(* CODESYS project WashingMashingProject_SimoneUtili.project

Project tree, tasks and I/O mapping:
  Device : CODESYS Control Win V3, CODESYS, version 3.5.20.0
    application Application
      libraries: Standard, 3.5.18.0 (System); VisuDialogs, * (System)
      task VISU_TASK (cyclic, interval 100 ms, priority 31) calls VisuElems.Visu_Prg
      task MainTask (cyclic, interval t#20ms, priority 1) calls ParentPolicyAutomata, Nominal_PA, WInFaulty_PA, HeatFaulty_PA, Simulation_Program, GA_Collector
      visualisation Visualization
      FUNCTIONBLOCKs/
        GAs/
          function block WaterManagement_GA [SFC]: _aSetDone_exit, _aEmptyWater_exit, _aFillWater_exit, _aInit_active, _aEmptyWater_active, _aReady_exit, _aReady_active, _aCHECKLEV_active, _aEmptyWater_entry, _aSetDone_active, _aFillWater_active, _aFillWater_entry_1
          function block TempControl_GA [SFC]: _aReady_exit, _aInit_active, _aReady_active, _aHeating_entry, _aHeating_exit, _aHeating_active
          function block DoorLocking_GA [SFC]: _aLocking_active, _aReady_active, _aInit_active, _aUnlocking_active, _aReady_exit, _aLocking_entry, _aUnlocking_entry, _aUnlocking_exit, _aLocking_exit, _aDoorCheck_active
          function block SoapEmptying_GA [SFC]: _aReady_active, _aCheckLev_active, _aReady_exit, _aInit_active, _aEmptying_active, _aEmptying_exit
          function block DrumMotor_GA [SFC]: _aBusy_active, _aReady_active, _aInit_active, _aBusy_exit
      PROGRAMs/
        program Simulation_Program [ST]
        program GA_Collector [FBD]
        Policy_Automatas/
          Child_PAs/
            program Nominal_PA [SFC]: _aCHECK_active, _aFLAGS_active, _aDoorLock_active_1, _aDoorLock_entry_1, _aDoorLock_exit_1, _aFillWater_active_1, _aFillWater_entry_1, _aFillWater_exit_1, _aTempRegON_active_1, _aStartMotor_active_1_1, _aStartMotSoap_active, _aStopMotor_active_1, _aStopMotor_exit_1, _aTempRegOFF_active_1, _aTempRegOFF_exit_1, _aEmptyWater_active_1, _aEmptyWater_exit_1, _aPhaseUpdate_active_1, _aPhaseUpdate_exit_1, _aDoorUnlock_active_1, _aDoorUnlock_exit_1, _aFinishedFlag_active_1, _aInit_active, _aDoorUnlock_entry, _aFinishedFlag_entry
            FaultManagerPAs/
              program HeatFaulty_PA [SFC]: _aDummy_exit, _aFillWater_h_active, _aMotON_h_active, _aMotON2_h_active, _aInit_exit, _aEmptyWater_h_exit, _aMotOFF_h_exit, _aPhaseUpdate_h_active, _aSoapON_h_active, _aEmptyWater_h_active, _aPhaseUpdate_h_exit, _aFillWater_h_entry, _aInit_active, _aMotOFF_h_active, _aFillWater_h_exit
              program WInFaulty_PA [SFC]: _aTempRegON_exit, _aTempOFF_w_active, _aInit_active, _aMotON_w_active, _aTempOFF_w_exit, _tLavaggio, _aStartMotor2_active, _aTempON_w_active, _aMotOFF_w_exit, _aTempON_w_entry, _aMotON2_w_entry, _tNoLavaggio, _aSoapOFF_w_exit, _aMotON2_w_active, _aSoapON_w_active, _aSoapOFF_w_active, _aMotOFF_w_active
          program ParentPolicyAutomata [SFC]: _aNominalPA_entry, _aPAController_entry, _aHLevDiagnostics_active, _aPAController_exit, _aPAUSE_Nom_active_1, _aDummy_active, _aPAUSE_Flt_active, _tMultiFaults, _tPauseRequest2, _aHeat_flt_entry, _aWaterIn_flt_entry, _aWaterIn_flt_exit, _tMultiFaults2, _aHeat_flt_exit, _tPauseRequest1, _aParentPAInit_active, _aPAController_active, _aStopHeatTest_exit, _aFillTest_active, _aPAUSE_Flt_entry, _aEmptyTest_exit, _aIDOLSTEP_entry, _aUnlockDoor_exit, _aRestore_exit, _aStartHeatTest_active, _aPAUSE_Nom_entry_1, _aFillTest_exit, _aStartHeatTest_entry, _aUnlockDoor_entry, _aIDOLSTEP_active, _aRestore_active, _aEmptyWater_exit, _aPAUSE_Nom_exit_1, _aStopHeatTest_active, _aEmptyWater_active, _aEmptyTest_active, _aFaultExpired_exit, _aPAUSE_Flt_exit, _aStartHeatTest_exit, _aUnlockDoor_active, _aNominalPA_exit, _tPauseRequest_
      FUNCTIONs/
        function SetBools [ST]
        function CheckFault [ST]
        function WMTempCheck [ST]
        function WMprogramCheck [ST]
        function FaultHMI [ST]
      Variables/
        ENUMs/
          data type WMPrograms
          data type State_FB
          data type Action_State
          data type LedStates
          data type LockerDoWhats
          data type WaterDoWhats
          data type WMTemps
          data type WInFlt_cases
          data type PolicyDegradation
          data type FaultType
          data type WashingPhase
        global variables GVL
  text list GlobalTextList
*)

// Device/Application/Variables/ENUMs/WMPrograms
//{attribute 'qualified_only'}
//{attribute 'strict'}
(*Programmi di funzionamento previsti dal comportamento nominale della lavatrice e selezionabili dall'utente*)
TYPE WMPrograms :
(
	Prelavaggio_prog := 1,
	Lavaggio_prog := 2,
	LavaggioCompleto_prog := 3
);
END_TYPE

// Device/Application/Variables/ENUMs/State_FB
//{attribute 'qualified_only'}
//{attribute 'strict'}

(*DUT enumerativo per definire lo stato presente della macchina a stati implementata nel SFC di ogni GA*)
TYPE State_FB : 
(
	S_Init := 0,
	S_Ready := 1,
	S_Busy := 2,
	S_Fault
);
END_TYPE

// Device/Application/Variables/ENUMs/Action_State
//{attribute 'qualified_only'}
//{attribute 'strict'}
(*stato della macchina a stati implementata nel SFC delle politiche durante il coordinamento di un GA*)
TYPE Action_State :
(
	Start_Action := 0,
	Wait_Compl := 1,
	SetOpOk := 2
);
END_TYPE

// Device/Application/Variables/ENUMs/LedStates
//{attribute 'qualified_only'}
//{attribute 'strict'}
(*due stati di accensione o spegnimento di un led*)
TYPE LedStates :
(
	ON := 0,
	OFF := 1
);
END_TYPE

// Device/Application/Variables/ENUMs/LockerDoWhats
//{attribute 'qualified_only'}
//{attribute 'strict'}
TYPE LockerDoWhats :
(
	Do_Locking := 0,
	Do_Unlocking :=1
);
END_TYPE

// Device/Application/Variables/ENUMs/WaterDoWhats
//{attribute 'qualified_only'}
//{attribute 'strict'}
TYPE WaterDoWhats :
(
	Do_WaterFilling := 0,
	Do_WaterEmptying := 1
);
END_TYPE

// Device/Application/Variables/ENUMs/WMTemps
//{attribute 'qualified_only'}
//{attribute 'strict'}

(*Temperature dell'acqua possibili selezionabili dall'utente*)
TYPE WMTemps :
(
	Warm30 := 30,
	Warm60 := 60,
	Warm90 := 90
);
END_TYPE

// Device/Application/Variables/ENUMs/WInFlt_cases
//{attribute 'qualified_only'}
//{attribute 'strict'}
(*variabile di uscita di interfaccia del GA di gestione dell'acqua per la fault isolation specifica dell'anomalia
WaterIn sulla base del livello di acqua presente nel cestello nel momento in cui il tubo si ottura*)
TYPE WInFlt_cases :
(
	early := 1,
	mid := 2,
	late := 3
);
END_TYPE

// Device/Application/Variables/ENUMs/PolicyDegradation
//{attribute 'qualified_only'}
//{attribute 'strict'}
(* Stato di salute della Politica in esecuzione*)
TYPE PolicyDegradation :
(
	HealthyPA := 0,
	FaultyPA := 1,
	KilledPA := 2
);
END_TYPE

// Device/Application/Variables/ENUMs/FaultType
//{attribute 'qualified_only'}
//{attribute 'strict'}
(*Tipo di fault riscontrato*)
TYPE FaultType :
(
	None := 0,
	WaterIn := 1,
	WaterOut := 2,
	Heat
);
END_TYPE

// Device/Application/Variables/ENUMs/WashingPhase
//{attribute 'qualified_only'}
//{attribute 'strict'}
(*Fasi di lavoro possibili per ogni programma di funzionamento della lavatrice*)
TYPE WashingPhase :
(
	Prelavaggio := 1,
	Lavaggio := 2,
	Risciacquo := 3,
	NOP
);
END_TYPE

// Device/Application/Variables/GVL
//{attribute 'qualified_only'}
VAR_GLOBAL
	temperature		: INT;		 	(*Sensor: current temperature of the water*)
	soaplevel		: INT; 			(*Sensor: current soap level*)
	waterlevel		: INT;			(*Sensor: current water level*)
	prog_number		: INT;			(*Input: program selected by the user*)
	temp_number		: INT; 			(*Input: temperature selected by the user*)
	run				: BOOL;			(*Input: if TRUE the washing machine works*)
	fillsoap		: BOOL; 		(*Input: if TRUE the soap tray is full*)
	bulls_eye_open	: BOOL := TRUE;	(*Input: if TRUE the door is open*)

	hot				: BOOL;			(*Actuator: if TRUE the resistor turns on*)
	motor_on		: BOOL;			(*Actuator: if TRUE the basket motor is turned on*)
	bulls_eye_lock	: BOOL;			(*Actuator: if TRUE the Door is locked*)
	emptysoap		: BOOL;			(*Actuator: if TRUE the soap tray is emptied*)
	fillwater		: BOOL;			(*Actuator: if TRUE the water is added*)
	emptywater		: BOOL;			(*Actuator: if TRUE the water is drained*)

	heat_alarm		: BOOL; 		(*Visualization: if TRUE alerts the user of the resistor fault*)
	water_in_alarm	: BOOL;			(*Visualization: if TRUE alerts the user of the water intake valve fault*)
	water_out_alarm	: BOOL; 		(*Visualization: if TRUE alerts the user of the water drain valve fault*)
	soap_alarm		: BOOL;			(*Visualization: if TRUE there is no soap*)
	prog_error		: BOOL;			(*Visualization: if TRUE the program selected is wrong*)
	temp_error		: BOOL;			(*Visualization: if TRUE the temperature selected is wrong*)
	rinse			: BOOL; 		(*Visualization: if TRUE the rinsing operation is going on*)
	prewash			: BOOL; 		(*Visualization: if TRUE the prewashing operation is going on*)
	wash			: BOOL; 		(*Visualization: if TRUE the washing operation is going on*)

	motor			: INT;			(*Only for simulation: angular position of the basket*)
	heat_fail		: BOOL;			(*Only for simulation: if TRUE the resistor cannot turn on*)
	water_in_fail	: BOOL;			(*Only for simulation: if TRUE the water intake valve is faulty*)
	water_out_fail	: BOOL;			(*Only for simulation: if TRUE the water drain valve is faulty*)
	WaterManagement_GA_0: WaterManagement_GA;
	TempControl_GA_0: TempControl_GA;
	SoapEmptying_GA_0: SoapEmptying_GA;
	DoorLocking_GA_0: DoorLocking_GA;
	DrumMotor_GA_0: DrumMotor_GA;
	SelectedProg : WMPrograms;
	SelectedTemp: WMTemps;
	Action_S: Action_State := Start_Action;
	Washing_P : WashingPhase;
	OpOk: BOOL;
	ProgDone: BOOL;
	IDOL : BOOL;
	PolicyEval: PolicyDegradation := HealthyPA; //inizializzo la policy come healthy per avere il comportamento nominale all'inizio
	WashTime: TIME;
	Do_Abort: BOOL;
END_VAR

// Device/Application/PROGRAMs/Policy_Automatas/ParentPolicyAutomata
PROGRAM ParentPolicyAutomata
VAR
	FltManag: BOOL := OpOk AND WaterManagement_GA_0.EmptyWaterOk;
	Fault: ARRAY [0..2] OF FaultType:= [None,None,None];
	RestoreTime : TIME := T#5S;
	Delay : TON;
	flashing : LedStates := ON;
	i:INT := 0;
END_VAR
(* SFC genitore per gestire l'esecuzione dei PA figli (Nominale, Faulty) e per eseguire gli step di attesa (IDOL), 
ripristino del funzionamento nominale e verifica delle riparazioni da fault*)

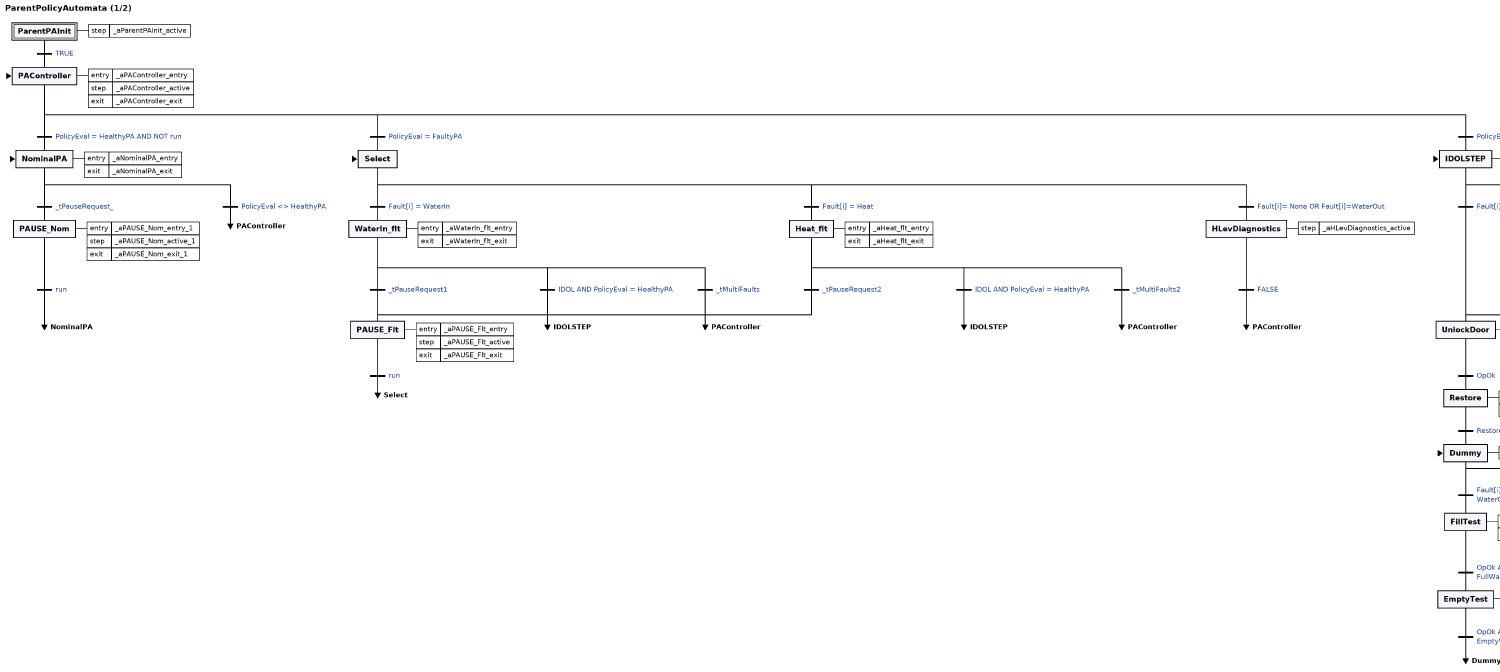
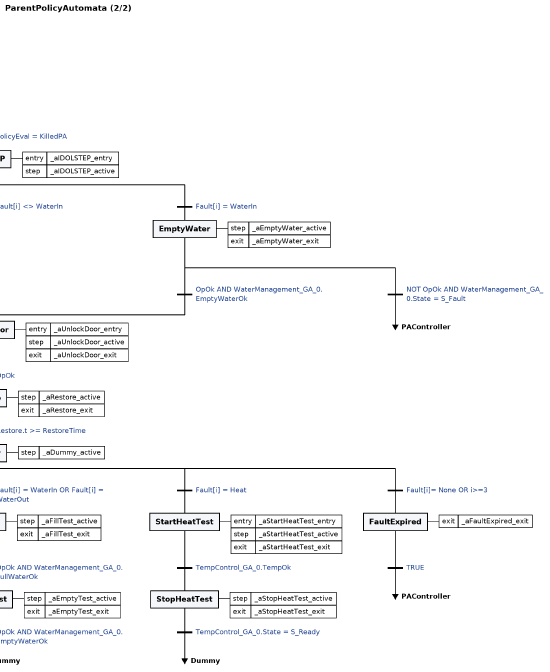
INITIAL_STEP ParentPAInit:
    _aParentPAInit_active(N);  // step action
END_STEP
TRANSITION FROM ParentPAInit TO PAController
    := TRUE;
END_TRANSITION
STEP PAController:
    _aPAController_entry(P1);  // entry action
    _aPAController_active(N);  // step action
    _aPAController_exit(P0);  // exit action
END_STEP
TRANSITION FROM PAController TO NominalPA
    := PolicyEval = HealthyPA AND NOT run;
END_TRANSITION
STEP NominalPA:
    _aNominalPA_entry(P1);  // entry action
    _aNominalPA_exit(P0);  // exit action
END_STEP
TRANSITION FROM NominalPA TO PAUSE_Nom
    := _tPauseRequest_;
END_TRANSITION
STEP PAUSE_Nom:
    _aPAUSE_Nom_entry_1(P1);  // entry action
    _aPAUSE_Nom_active_1(N);  // step action
    _aPAUSE_Nom_exit_1(P0);  // exit action
END_STEP
TRANSITION FROM PAUSE_Nom TO NominalPA
    := run;
END_TRANSITION
TRANSITION FROM NominalPA TO PAController
    := PolicyEval <> HealthyPA;
END_TRANSITION
TRANSITION FROM PAController TO Select
    := PolicyEval = FaultyPA;
END_TRANSITION
// macro FaultyPAs begins
STEP Select:
END_STEP
TRANSITION FROM Select TO WaterIn_flt
    := Fault[i] = WaterIn;
END_TRANSITION
STEP WaterIn_flt:
    _aWaterIn_flt_entry(P1);  // entry action
    _aWaterIn_flt_exit(P0);  // exit action
END_STEP
TRANSITION FROM WaterIn_flt TO PAUSE_Flt
    := _tPauseRequest1;
END_TRANSITION
TRANSITION FROM WaterIn_flt TO IDOLSTEP
    := IDOL AND PolicyEval = HealthyPA;
END_TRANSITION
TRANSITION FROM WaterIn_flt TO PAController
    := _tMultiFaults;
END_TRANSITION
TRANSITION FROM Select TO Heat_flt
    := Fault[i] = Heat;
END_TRANSITION
STEP Heat_flt:
    _aHeat_flt_entry(P1);  // entry action
    _aHeat_flt_exit(P0);  // exit action
END_STEP
TRANSITION FROM Heat_flt TO PAUSE_Flt
    := _tPauseRequest2;
END_TRANSITION
TRANSITION FROM Heat_flt TO IDOLSTEP
    := IDOL AND PolicyEval = HealthyPA;
END_TRANSITION
TRANSITION FROM Heat_flt TO PAController
    := _tMultiFaults2;
END_TRANSITION
TRANSITION FROM Select TO HLevDiagnostics
    := Fault[i]= None OR Fault[i]=WaterOut;
END_TRANSITION
STEP HLevDiagnostics:
    _aHLevDiagnostics_active(N);  // step action
END_STEP
TRANSITION FROM HLevDiagnostics TO PAController
    := FALSE;
END_TRANSITION
STEP PAUSE_Flt:
    _aPAUSE_Flt_entry(P1);  // entry action
    _aPAUSE_Flt_active(N);  // step action
    _aPAUSE_Flt_exit(P0);  // exit action
END_STEP
TRANSITION FROM PAUSE_Flt TO Select
    := run;
END_TRANSITION
TRANSITION FROM PAController TO IDOLSTEP
    := PolicyEval = KilledPA;
END_TRANSITION
// macro IdolAndTest begins
STEP IDOLSTEP:
    _aIDOLSTEP_entry(P1);  // entry action
    _aIDOLSTEP_active(N);  // step action
END_STEP
TRANSITION FROM IDOLSTEP TO UnlockDoor
    := Fault[i] <> WaterIn;
END_TRANSITION
TRANSITION FROM IDOLSTEP TO EmptyWater
    := Fault[i] = WaterIn;
END_TRANSITION
STEP EmptyWater:
    _aEmptyWater_active(N);  // step action
    _aEmptyWater_exit(P0);  // exit action
END_STEP
TRANSITION FROM EmptyWater TO UnlockDoor
    := OpOk AND WaterManagement_GA_0.EmptyWaterOk;
END_TRANSITION
TRANSITION FROM EmptyWater TO PAController
    := NOT OpOk AND WaterManagement_GA_0.State = S_Fault;
END_TRANSITION
STEP UnlockDoor:
    _aUnlockDoor_entry(P1);  // entry action
    _aUnlockDoor_active(N);  // step action
    _aUnlockDoor_exit(P0);  // exit action
END_STEP
TRANSITION FROM UnlockDoor TO Restore
    := OpOk;
END_TRANSITION
STEP Restore:
    _aRestore_active(N);  // step action
    _aRestore_exit(P0);  // exit action
END_STEP
TRANSITION FROM Restore TO Dummy
    := Restore.t >= RestoreTime;
END_TRANSITION
STEP Dummy:
    _aDummy_active(N);  // step action
END_STEP
TRANSITION FROM Dummy TO FillTest
    := Fault[i] = WaterIn OR Fault[i] = WaterOut;
END_TRANSITION
STEP FillTest:
    _aFillTest_active(N);  // step action
    _aFillTest_exit(P0);  // exit action
END_STEP
TRANSITION FROM FillTest TO EmptyTest
    := OpOk AND WaterManagement_GA_0.FullWaterOk;
END_TRANSITION
STEP EmptyTest:
    _aEmptyTest_active(N);  // step action
    _aEmptyTest_exit(P0);  // exit action
END_STEP
TRANSITION FROM EmptyTest TO Dummy
    := OpOk AND WaterManagement_GA_0.EmptyWaterOk;
END_TRANSITION
TRANSITION FROM Dummy TO StartHeatTest
    := Fault[i] = Heat;
END_TRANSITION
STEP StartHeatTest:
    _aStartHeatTest_entry(P1);  // entry action
    _aStartHeatTest_active(N);  // step action
    _aStartHeatTest_exit(P0);  // exit action
END_STEP
TRANSITION FROM StartHeatTest TO StopHeatTest
    := TempControl_GA_0.TempOk;
END_TRANSITION
STEP StopHeatTest:
    _aStopHeatTest_active(N);  // step action
    _aStopHeatTest_exit(P0);  // exit action
END_STEP
TRANSITION FROM StopHeatTest TO Dummy
    := TempControl_GA_0.State = S_Ready;
END_TRANSITION
TRANSITION FROM Dummy TO FaultExpired
    := Fault[i]= None OR i>=3;
END_TRANSITION
STEP FaultExpired:
    _aFaultExpired_exit(P0);  // exit action
END_STEP
TRANSITION FROM FaultExpired TO PAController
    := TRUE;
END_TRANSITION

ACTION _aNominalPA_entry:
WashTime := T#5S;
Nominal_PA.SFCInit := FALSE;
END_ACTION

ACTION _aPAController_entry:
IF Fault[i] <> None THEN
	i:=i+1;
END_IF
END_ACTION

ACTION _aHLevDiagnostics_active:
//Questo step rappresenta una diagnositica di alto livello di tipo A per l'interfacciamento corretto tra Politica e GA

(*Nota: questo step non dovrebbe essere mai eseguito perchè il ramo di PAFaulty viene attraversato solo nel 
caso di WaterIn o Heat fault, per nessun Fault dovrebbe essere attivo l'SFC Nominale o la fase di IdolAndStep 
nel caso di fault già gestiti*)
END_ACTION

ACTION _aPAController_exit:
FaultHMI(Fault[i], TRUE);

IF Fault[i]= None THEN
 SetBools(3,FALSE);
END_IF
END_ACTION

ACTION _aPAUSE_Nom_active_1:

END_ACTION

ACTION _aDummy_active:
//step con nessuna aziona per permettere un loop corretto dei fault nel vettore che li contiene

(*Una volta avvvenuto l'intervento di ripristino degli attuatori malfunzionanti, prima di procedere con 
un programma inserito dall'utente si fa un test delle azioni base relative all'attuatore che è stato riparato
per verificare il corretto intervento*)
END_ACTION

ACTION _aPAUSE_Flt_active:

END_ACTION

TRANSITION _tMultiFaults:
PolicyEval <> HealthyPA AND WaterManagement_GA_0.State = S_Ready
END_TRANSITION

TRANSITION _tPauseRequest2:
PolicyEval = HealthyPA AND NOT run
END_TRANSITION

ACTION _aHeat_flt_entry:
HeatFaulty_PA.SFCInit := FALSE;
TempControl_GA_0.StartTemp := FALSE;

//Le seguenti sono istruzioni per garantire un protocollo di handshake corretto tra Parent Policy e Child Policy
//Esco dallo stato di fault in modo da riconoscere un'eventuale condizione di fault aggiuntivo (fault multipli)
//durante l'esecuzione degradata del programma dovuta al primo fault
 
TempControl_GA_0.Restore := TRUE; //PER ANDARE IN READY NEL GA
WashTime := T#3S;
END_ACTION

ACTION _aWaterIn_flt_entry:
WInFaulty_PA.SFCInit := FALSE;
WaterManagement_GA_0.Restore := TRUE;
END_ACTION

ACTION _aWaterIn_flt_exit:
WInFaulty_PA.SFCPause := TRUE;

//WInFaulty_PA.SFCInit := TRUE;
WaterManagement_GA_0.Restore := FALSE;
END_ACTION

TRANSITION _tMultiFaults2:
PolicyEval <> HealthyPA AND TempControl_GA_0.State = S_Ready

//Se la politica non è più Healthy durante l'esecuzione dell'AdP HeatFaulty_PA allora
//significa che è avvenuto un altro fault
END_TRANSITION

ACTION _aHeat_flt_exit:
HeatFaulty_PA.SFCPause := TRUE;
HeatFaulty_PA.SFCInit := TRUE;
TempControl_GA_0.Restore := FALSE;
END_ACTION

TRANSITION _tPauseRequest1:
PolicyEval = HealthyPA AND NOT run
END_TRANSITION

ACTION _aParentPAInit_active:

END_ACTION

ACTION _aPAController_active:
SetBools(4,TRUE); //inizializzo le SFC Flags
IF NOT IDOL  THEN
	Fault[i] := checkFault();
END_IF
END_ACTION

ACTION _aStopHeatTest_exit:
TempControl_GA_0.StopTemp := FALSE;
i:=i+1;
END_ACTION

ACTION _aFillTest_active:
CASE Action_S OF 
Start_Action: IF WaterManagement_GA_0.State = S_Ready THEN 
				 WaterManagement_GA_0.FillTest := TRUE;
				 Action_S := Wait_Compl;
			  END_IF
			  
Wait_Compl: IF WaterManagement_GA_0.Done AND WaterManagement_GA_0.State = S_Busy THEN 
			   WaterManagement_GA_0.FillTest := FALSE;
			   Action_S := SetOpOk;
			END_IF
//protocollo di handshake di set reset del FillTest e done da parte di politica e ga per evitare attivazioni multiple
SetOpOk: IF NOT WaterManagement_GA_0.Done THEN
			OpOk := TRUE;
	     END_IF
END_CASE
END_ACTION

ACTION _aPAUSE_Flt_entry:
Do_Abort := TRUE;
SetBools(2,FALSE);
END_ACTION

ACTION _aEmptyTest_exit:
OpOk := FALSE;
Action_S := Start_Action;
i:=i+1;
END_ACTION

ACTION _aIDOLSTEP_entry:
IDOL := FALSE;
WaterManagement_GA_0.Restore := TRUE;
END_ACTION

ACTION _aUnlockDoor_exit:
OpOk := FALSE;
Action_S := Start_Action;
END_ACTION

ACTION _aRestore_exit:
SetBools(3,FALSE);
i:=0;
END_ACTION

ACTION _aStartHeatTest_active:
IF TempControl_GA_0.State = S_Ready THEN
	TempControl_GA_0.StartWhat := Warm90;
	TempControl_GA_0.HeatTest := TRUE;
END_IF
END_ACTION

ACTION _aPAUSE_Nom_entry_1:
Do_Abort := TRUE;
SetBools(2,FALSE);
END_ACTION

ACTION _aFillTest_exit:
OpOk := FALSE;
Action_S := Start_Action;
END_ACTION

ACTION _aStartHeatTest_entry:
TempControl_GA_0.StopTemp := FALSE; //protocollo di handshake per evitare attivazioni multiple
END_ACTION

ACTION _aUnlockDoor_entry:
Action_S := Start_Action;
WaterManagement_GA_0.Restore := FALSE;
END_ACTION

ACTION _aIDOLSTEP_active:
SetBools(2,FALSE); //spegnimento led fasi hmi nel caso di un fault killer
END_ACTION

ACTION _aRestore_active:
//IMPORTANTE!!
(*Questo è lo step in cui si ipotizza avvenga l'intervento da parte di un operatore esterno per eseguire la manutenzione
necessaria al ripristino del funzionamento nominale della lavatrice e delle sue funzioni, per semplicità si considera
che l'intervento avvenga senza disalimentare la lavatrice e gli attuatori stessi, nella simulazione perciò
si spengono gli switch dei fault durante questa fase caratterizzata dal lampeggiamento dei led hmi dei fault riscontrati
*)
CASE flashing OF 
ON: FaultHMI(Fault[0], FALSE);
	FaultHMI(Fault[1], FALSE);
	FaultHMI(Fault[2],FALSE);
	Delay(IN:=TRUE, PT:=T#0.3S);
	IF Delay.Q THEN
		Delay(IN:=FALSE);
		flashing := OFF;
	END_IF
OFF:FaultHMI(Fault[0], TRUE);
	FaultHMI(Fault[1], TRUE);
	FaultHMI(Fault[2],TRUE);
	Delay(IN:=TRUE, PT:=T#0.3S);
	IF Delay.Q THEN
	  Delay(IN:=FALSE); 
	  flashing := ON;
	END_IF
END_CASE
END_ACTION

ACTION _aEmptyWater_exit:
OpOk := FALSE;
Action_S := Start_Action;
END_ACTION

ACTION _aPAUSE_Nom_exit_1:
Nominal_PA.SFCPause := FALSE;
Do_Abort := FALSE;

CASE Washing_P OF 
Prelavaggio: prewash := TRUE;
Lavaggio: wash := TRUE;
Risciacquo: rinse := TRUE;
END_CASE
END_ACTION

ACTION _aStopHeatTest_active:
TempControl_GA_0.StopTemp := TRUE;
TempControl_GA_0.StartTemp := FALSE;
TempControl_GA_0.HeatTest := FALSE;
END_ACTION

ACTION _aEmptyWater_active:
(* Nel caso di fault di tipo WaterIn si è scelto di svuotare l'acqua del cestello in questo step al termine della gestione che invece risulta differenziata
a seconda del momento in cui si interrompe il riempimento*)

CASE Action_S OF 
Start_Action: IF WaterManagement_GA_0.State = S_Ready THEN 
				 WaterManagement_GA_0.Do_ := TRUE;
				 WaterManagement_GA_0.DoWhat := Do_WaterEmptying;
				 Action_S := Wait_Compl;
			  END_IF
			  
Wait_Compl: IF WaterManagement_GA_0.Done AND WaterManagement_GA_0.State = S_Busy THEN 
			   WaterManagement_GA_0.Do_ := FALSE;
			   Action_S := SetOpOk;
			ELSIF NOT WaterManagement_GA_0.Done AND WaterManagement_GA_0.State = S_Fault THEN 
				WaterManagement_GA_0.Do_ := FALSE;
				Action_S := Start_Action;
			END_IF
//protocollo di handshake di set reset del do e done da parte di politica e ga per evitare attivazioni multiple
SetOpOk: IF NOT WaterManagement_GA_0.Done THEN
			OpOk := TRUE;
	     END_IF
END_CASE
END_ACTION

ACTION _aEmptyTest_active:
CASE Action_S OF 
Start_Action: IF WaterManagement_GA_0.State = S_Ready THEN 
				 //WaterManagement_GA_0.Do_ := TRUE;
				 //WaterManagement_GA_0.DoWhat := Do_WaterEmptying;
				 WaterManagement_GA_0.EmptyTest := TRUE;
				 Action_S := Wait_Compl;
			  END_IF
			  
Wait_Compl: IF WaterManagement_GA_0.Done AND WaterManagement_GA_0.State = S_Busy THEN 
			   //WaterManagement_GA_0.Do_ := FALSE;
			   WaterManagement_GA_0.EmptyTest := FALSE;
			   Action_S := SetOpOk;
			END_IF
//protocollo di handshake di set reset del do e done da parte di politica e ga per evitare attivazioni multiple
SetOpOk: IF NOT WaterManagement_GA_0.Done THEN
			OpOk := TRUE;
	     END_IF
END_CASE
END_ACTION

ACTION _aFaultExpired_exit:
//tutti i fault sono estinti e ne è stata verificata l'assenza in seguito all'intervento dell'operatore

//inizializzo i parametri di gestione dei fault per ricominciare un altro programma di lavaggio
//della lavatrice a partire dalla Politica Nominale
i:=0;
PolicyEval := HealthyPA;
Washing_P := NOP;
Fault[0]:= None;
Fault[1]:= None;
Fault[2] := None;
END_ACTION

ACTION _aPAUSE_Flt_exit:
WInFaulty_PA.SFCPause := FALSE;
HeatFaulty_PA.SFCPause := FALSE;
Do_Abort := FALSE;

CASE Washing_P OF 
Prelavaggio: prewash := TRUE;
Lavaggio: wash := TRUE;
Risciacquo: rinse := TRUE;
END_CASE
END_ACTION

ACTION _aStartHeatTest_exit:

END_ACTION

ACTION _aUnlockDoor_active:
CASE Action_S OF 
Start_Action: IF Doorlocking_GA_0.State = S_Ready THEN 
				 Doorlocking_GA_0.Do_ := TRUE;
				 Doorlocking_GA_0.DoWhat := Do_Unlocking;
				 Action_S := Wait_Compl;
			  END_IF
			  
Wait_Compl: IF Doorlocking_GA_0.Done AND Doorlocking_GA_0.State = S_Busy THEN 
			   Doorlocking_GA_0.Do_ := FALSE;
			   Action_S := SetOpOk;
			END_IF
//protocollo di handshake di set reset del do e done da parte di politica e ga per evitare attivazioni multiple
SetOpOk: IF NOT Doorlocking_GA_0.Done THEN
			OpOk := TRUE;
	     END_IF
END_CASE
END_ACTION

ACTION _aNominalPA_exit:
Nominal_PA.SFCPause := TRUE;
END_ACTION

TRANSITION _tPauseRequest_:
PolicyEval = HealthyPA AND NOT run
END_TRANSITION

END_PROGRAM

// Device/Application/PROGRAMs/Policy_Automatas/Child_PAs/Nominal_PA
PROGRAM Nominal_PA
VAR
	TempCorrect: BOOL;
	ProgCorrect: BOOL;
	SoapCorrect: BOOL;
	LockCorrect: BOOL;
	CheckOk: BOOL;
	Delay : TON;
	flashing : LedStates := ON;
END_VAR
VAR_INPUT
	SFCInit:BOOL;
	SFCPause: BOOL;
END_VAR

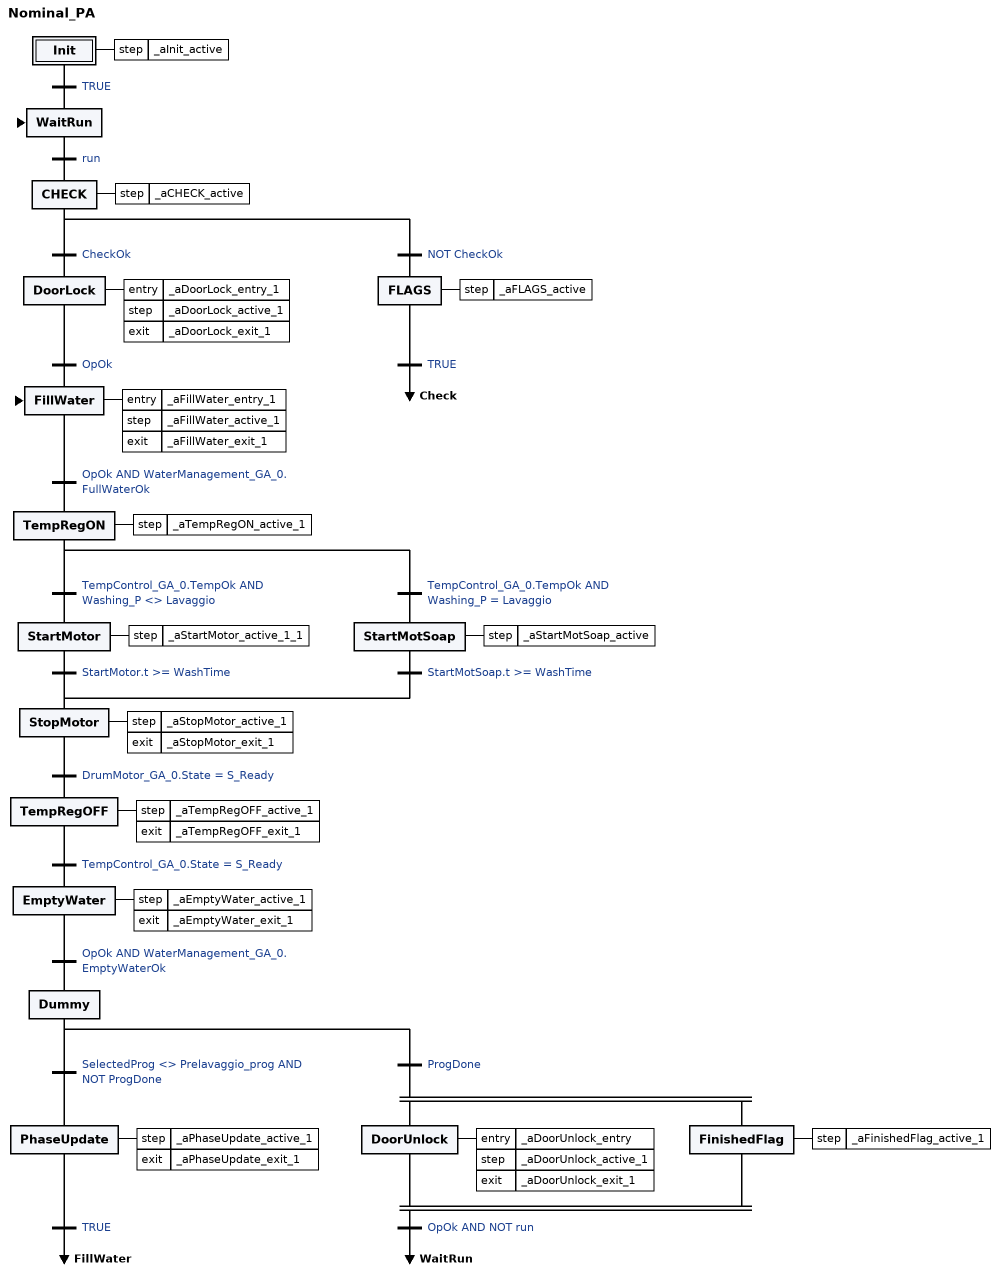
INITIAL_STEP Init:
    _aInit_active(N);  // step action
END_STEP
TRANSITION FROM Init TO WaitRun
    := TRUE;
END_TRANSITION
STEP WaitRun:
END_STEP
TRANSITION FROM WaitRun TO CHECK
    := run;
END_TRANSITION
STEP CHECK:
    _aCHECK_active(N);  // step action
END_STEP
TRANSITION FROM CHECK TO DoorLock
    := CheckOk;
END_TRANSITION
// macro WMCYCLE begins
STEP DoorLock:
    _aDoorLock_entry_1(P1);  // entry action
    _aDoorLock_active_1(N);  // step action
    _aDoorLock_exit_1(P0);  // exit action
END_STEP
TRANSITION FROM DoorLock TO FillWater
    := OpOk;
END_TRANSITION
STEP FillWater:
    _aFillWater_entry_1(P1);  // entry action
    _aFillWater_active_1(N);  // step action
    _aFillWater_exit_1(P0);  // exit action
END_STEP
TRANSITION FROM FillWater TO TempRegON
    := OpOk AND WaterManagement_GA_0.FullWaterOk;
END_TRANSITION
STEP TempRegON:
    _aTempRegON_active_1(N);  // step action
END_STEP
TRANSITION FROM TempRegON TO StartMotor
    := TempControl_GA_0.TempOk AND Washing_P <> Lavaggio;
END_TRANSITION
STEP StartMotor:
    _aStartMotor_active_1_1(N);  // step action
END_STEP
TRANSITION FROM StartMotor TO StopMotor
    := StartMotor.t >= WashTime;
END_TRANSITION
TRANSITION FROM TempRegON TO StartMotSoap
    := TempControl_GA_0.TempOk AND Washing_P = Lavaggio;
END_TRANSITION
STEP StartMotSoap:
    _aStartMotSoap_active(N);  // step action
END_STEP
TRANSITION FROM StartMotSoap TO StopMotor
    := StartMotSoap.t >= WashTime;
END_TRANSITION
STEP StopMotor:
    _aStopMotor_active_1(N);  // step action
    _aStopMotor_exit_1(P0);  // exit action
END_STEP
TRANSITION FROM StopMotor TO TempRegOFF
    := DrumMotor_GA_0.State = S_Ready;
END_TRANSITION
STEP TempRegOFF:
    _aTempRegOFF_active_1(N);  // step action
    _aTempRegOFF_exit_1(P0);  // exit action
END_STEP
TRANSITION FROM TempRegOFF TO EmptyWater
    := TempControl_GA_0.State = S_Ready;
END_TRANSITION
STEP EmptyWater:
    _aEmptyWater_active_1(N);  // step action
    _aEmptyWater_exit_1(P0);  // exit action
END_STEP
TRANSITION FROM EmptyWater TO Dummy
    := OpOk AND WaterManagement_GA_0.EmptyWaterOk;
END_TRANSITION
STEP Dummy:
END_STEP
TRANSITION FROM Dummy TO PhaseUpdate
    := SelectedProg <> Prelavaggio_prog AND NOT ProgDone;
END_TRANSITION
STEP PhaseUpdate:
    _aPhaseUpdate_active_1(N);  // step action
    _aPhaseUpdate_exit_1(P0);  // exit action
END_STEP
TRANSITION FROM PhaseUpdate TO FillWater
    := TRUE;
END_TRANSITION
TRANSITION FROM Dummy TO (DoorUnlock, FinishedFlag)
    := ProgDone;
END_TRANSITION
STEP DoorUnlock:
    _aDoorUnlock_entry(P1);  // entry action
    _aDoorUnlock_active_1(N);  // step action
    _aDoorUnlock_exit_1(P0);  // exit action
END_STEP
STEP FinishedFlag:
    _aFinishedFlag_active_1(N);  // step action
END_STEP
TRANSITION FROM (DoorUnlock, FinishedFlag) TO WaitRun
    := OpOk AND NOT run;
END_TRANSITION
TRANSITION FROM CHECK TO FLAGS
    := NOT CheckOk;
END_TRANSITION
STEP FLAGS:
    _aFLAGS_active(N);  // step action
END_STEP
TRANSITION FROM FLAGS TO Check
    := TRUE;
END_TRANSITION

ACTION _aCHECK_active:
//Per la corretta gestione dell'HMI mplementa il freeze delle variabili da hmi 
//vengono cioè salvati i primi input non più modificabili se non in un secondo ciclo di check nel programma successivo
SelectedProg := prog_number; //int to type enum
SelectedTemp := temp_number;

ProgCorrect := WMProgramCheck(SelectedProg);
TempCorrect := WMTempCheck(SelectedTemp);

IF ProgCorrect THEN
	CASE SelectedProg OF 
	Prelavaggio_prog: SoapCorrect := TRUE; //l'unico programma che non richiede il sapone è il prelavaggio perciò il check è già verificato
		Washing_P := Prelavaggio; //inilizializzazione della prima fase corrispondente al programma selezionato
		ProgDone := TRUE; //non richiede loop
		
	Lavaggio_prog: IF NOT SoapEmptying_GA_0.NoSoap THEN 
			SoapCorrect := TRUE;
		ELSE 	SoapCorrect := FALSE;
		END_IF 
	   Washing_P := Lavaggio;
	   
	LavaggioCompleto_prog: IF NOT SoapEmptying_GA_0.NoSoap THEN 
			SoapCorrect := TRUE;
		ELSE 	SoapCorrect := FALSE;
		END_IF 
	   Washing_P := Prelavaggio;
	   
	END_CASE
END_IF

IF NOT DoorLocking_GA_0.OpenDoor THEN
	LockCorrect := TRUE;
END_IF

//check delle variabili di input contemporaneamente
IF TempCorrect AND ProgCorrect AND SoapCorrect AND LockCorrect THEN 
	CheckOK := TRUE;
ELSE 
	CheckOk := FALSE;
END_IF
END_ACTION

ACTION _aFLAGS_active:
//led hmi segnalazione errore di input
soap_alarm := NOT SoapCorrect;
prog_error := NOT ProgCorrect;
temp_error := NOT TempCorrect;
END_ACTION

ACTION _aDoorLock_active_1:
CASE Action_S OF 
Start_Action: IF Doorlocking_GA_0.State = S_Ready THEN 
				 Doorlocking_GA_0.Do_ := TRUE;
				 Doorlocking_GA_0.DoWhat := Do_Locking;
				 Action_S := Wait_Compl;
			  END_IF
			  
Wait_Compl: IF Doorlocking_GA_0.Done AND Doorlocking_GA_0.State = S_Busy THEN 
			   Doorlocking_GA_0.Do_ := FALSE;
			   Action_S := SetOpOk;
			END_IF
//protocollo di handshake di set reset del do e done da parte di politica e ga per evitare attivazioni multiple
SetOpOk: IF NOT Doorlocking_GA_0.Done THEN
			OpOk := TRUE;
	     END_IF
END_CASE
END_ACTION

ACTION _aDoorLock_entry_1:
SetBools(1,FALSE); 
//spengono tutti i led di segnalazione di errori di input da hmi
//il primo parametro è il gruppo di variabili booleane da cambiare
END_ACTION

ACTION _aDoorLock_exit_1:
OpOk := FALSE;
Action_S := Start_Action;
END_ACTION

ACTION _aFillWater_active_1:
CASE Action_S OF //macchina a stati implementata con uno switch case, funziona grazie al modello di esecuzione con while intrinseco
//n.b. per fare la diagnostica di alto livello di tipo A tra politica e GA dovrei aggiungere un else nell'if per il caso il cui non si ver
//verifica mai lo stato ready(anomalia)
Start_Action: IF WaterManagement_GA_0.State = S_Ready THEN 
				 WaterManagement_GA_0.Do_ := TRUE;
				 WaterManagement_GA_0.DoWhat := Do_WaterFilling;
				 Action_S := Wait_Compl;
			  END_IF
			  
Wait_Compl: IF WaterManagement_GA_0.Done AND WaterManagement_GA_0.State = S_Busy THEN 
			   WaterManagement_GA_0.Do_ := FALSE;
			   Action_S := SetOpOk;
			   //nel caso di fault state del GA resetto il Do e inizializzo la macchina a stati
			ELSIF NOT WaterManagement_GA_0.Done AND WaterManagement_GA_0.State = S_Fault THEN 
				WaterManagement_GA_0.Do_ := FALSE;
				Action_S := Start_Action;
			END_IF
//protocollo di handshake di set reset del do e done da parte di politica e ga per evitare attivazioni multiple
SetOpOk: IF NOT WaterManagement_GA_0.Done THEN
			OpOk := TRUE;
	     END_IF
END_CASE
END_ACTION

ACTION _aFillWater_entry_1:

	CASE Washing_P OF 
	Prelavaggio: prewash := TRUE;
	Lavaggio: wash := TRUE;
	Risciacquo: rinse := TRUE;
	END_CASE
END_ACTION

ACTION _aFillWater_exit_1:
OpOk := FALSE;
Action_S := Start_Action;
END_ACTION

ACTION _aTempRegON_active_1:
IF TempControl_GA_0.State = S_Ready THEN
	TempControl_GA_0.StartWhat := SelectedTemp;
	TempControl_GA_0.StartTemp := TRUE;
END_IF
END_ACTION

ACTION _aStartMotor_active_1_1:
IF DrumMotor_GA_0.State = S_Ready THEN
	DrumMotor_GA_0.StartMotor := TRUE;
END_IF
END_ACTION

ACTION _aStartMotSoap_active:
IF DrumMotor_GA_0.State = S_Ready THEN
	DrumMotor_GA_0.StartMotor := TRUE;
END_IF

IF SoapEmptying_GA_0.State = S_Ready THEN
	SoapEmptying_GA_0.StartSoap := TRUE;
END_IF
END_ACTION

ACTION _aStopMotor_active_1:
DrumMotor_GA_0.StopMotor := TRUE;
DrumMotor_GA_0.StartMotor := FALSE;

SoapEmptying_GA_0.StopSoap := TRUE;
SoapEmptying_GA_0.StartSoap := FALSE;
END_ACTION

ACTION _aStopMotor_exit_1:
DrumMotor_GA_0.StopMotor := FALSE;
SoapEmptying_GA_0.StopSoap := FALSE;
END_ACTION

ACTION _aTempRegOFF_active_1:
TempControl_GA_0.StopTemp := TRUE;
TempControl_GA_0.StartTemp := FALSE;
END_ACTION

ACTION _aTempRegOFF_exit_1:
TempControl_GA_0.StopTemp := FALSE;
END_ACTION

ACTION _aEmptyWater_active_1:
CASE Action_S OF //macchina a stati implementata con uno switch case, funziona grazie al modello di esecuzione con while intrinseco
//n.b. per fare la diagnostica di alto livello di tipo A tra politica e GA dovrei aggiungere un else nell'if per il caso il cui non si ver
//verifica mai lo stato ready(anomalia)
Start_Action: IF WaterManagement_GA_0.State = S_Ready THEN 
				 WaterManagement_GA_0.Do_ := TRUE;
				 WaterManagement_GA_0.DoWhat := Do_WaterEmptying;
				 Action_S := Wait_Compl;
			  END_IF
			  
Wait_Compl: IF WaterManagement_GA_0.Done AND WaterManagement_GA_0.State = S_Busy THEN 
			   WaterManagement_GA_0.Do_ := FALSE;
			   Action_S := SetOpOk;
			 ELSIF NOT WaterManagement_GA_0.Done AND WaterManagement_GA_0.State = S_Fault THEN 
			   WaterManagement_GA_0.Do_ := FALSE;
			   Action_S := Start_Action;
			END_IF
//protocollo di handshake di set reset del do e done da parte di politica e ga per evitare attivazioni multiple
SetOpOk: IF NOT WaterManagement_GA_0.Done THEN
			OpOk := TRUE;
	     END_IF
END_CASE
END_ACTION

ACTION _aEmptyWater_exit_1:
OpOk := FALSE;
Action_S := Start_Action;
END_ACTION

ACTION _aPhaseUpdate_active_1:
IF SelectedProg = LavaggioCompleto_prog THEN
	CASE Washing_P OF 
	Prelavaggio: Washing_P := Lavaggio;
	
	Lavaggio : Washing_P := Risciacquo;
			   ProgDone := TRUE;
	END_CASE
END_IF

IF SelectedProg = Lavaggio_prog AND Washing_P = Lavaggio THEN
	Washing_P := Risciacquo;
	ProgDone := TRUE;
END_IF
END_ACTION

ACTION _aPhaseUpdate_exit_1:
prewash := FALSE;
wash := FALSE;
rinse := FALSE;
END_ACTION

ACTION _aDoorUnlock_active_1:

CASE Action_S OF 
Start_Action: IF Doorlocking_GA_0.State = S_Ready THEN 
				 Doorlocking_GA_0.Do_ := TRUE;
				 Doorlocking_GA_0.DoWhat := Do_Unlocking;
				 Action_S := Wait_Compl;
			  END_IF
			  
Wait_Compl: IF Doorlocking_GA_0.Done AND Doorlocking_GA_0.State = S_Busy THEN 
			   Doorlocking_GA_0.Do_ := FALSE;
			   Action_S := SetOpOk;
			END_IF
//protocollo di handshake di set reset del do e done da parte di politica e ga per evitare attivazioni multiple
SetOpOk: IF NOT Doorlocking_GA_0.Done THEN
			OpOk := TRUE;
	     END_IF
END_CASE
END_ACTION

ACTION _aDoorUnlock_exit_1:
OpOk := FALSE;
ProgDone := FALSE;
Action_S := Start_Action;
END_ACTION

ACTION _aFinishedFlag_active_1:
CASE flashing OF 
ON: SetBools(2,TRUE);
	Delay(IN:=TRUE, PT:=T#1S);
	IF Delay.Q THEN
		Delay(IN:=FALSE);
		flashing := OFF;
	END_IF
OFF: SetBools(2,FALSE);
	Delay(IN:=TRUE, PT:=T#1S);
	IF Delay.Q THEN
	  Delay(IN:=FALSE); 
	  flashing := ON;
	END_IF
END_CASE
END_ACTION

ACTION _aInit_active:
Washing_P := NOP;
END_ACTION

ACTION _aDoorUnlock_entry:
Washing_P := NOP;
END_ACTION

ACTION _aFinishedFlag_entry:

END_ACTION

END_PROGRAM

// Device/Application/FUNCTIONs/WMprogramCheck
FUNCTION WMprogramCheck : BOOL
VAR_INPUT
	InputProg : WMPrograms;
END_VAR
VAR
END_VAR

WMprogramCheck := InputProg = Prelavaggio_prog OR InputProg = Lavaggio_prog OR InputProg = LavaggioCompleto_prog;

END_FUNCTION

// Device/Application/FUNCTIONs/WMTempCheck
FUNCTION WMTempCheck : BOOL
VAR_INPUT
	InputTemp: WMTemps;
END_VAR
VAR
END_VAR

WMTempCheck := InputTemp = Warm30 OR InputTemp = Warm60 OR InputTemp = Warm90;

END_FUNCTION

// Device/Application/FUNCTIONs/SetBools
FUNCTION SetBools : BOOL
VAR_INPUT
	which: INT;
	value: BOOL;
END_VAR
VAR
END_VAR

CASE which OF 
	1:  prog_error := value;
		temp_error := value;
		soap_alarm := value;
		
	2:  prewash := value;
		wash := value;
		rinse := value;
		
	3:  water_in_alarm := value;
		water_out_alarm := value;
		heat_alarm := value;
		
	4:	Nominal_PA.SFCInit := value;
		WInFaulty_PA.SFCInit := value;
		HeatFaulty_PA.SFCInit := value;
		Nominal_PA.SFCPause := NOT value;
		WINFaulty_PA.SFCPause := NOT value;
		HeatFaulty_PA.SFCPause := NOT value;
	
END_CASE

END_FUNCTION

// Device/Application/PROGRAMs/Policy_Automatas/Child_PAs/FaultManagerPAs/WInFaulty_PA
PROGRAM WInFaulty_PA
VAR
END_VAR
VAR_INPUT
	SFCInit:BOOL;
	SFCPause: BOOL;
END_VAR

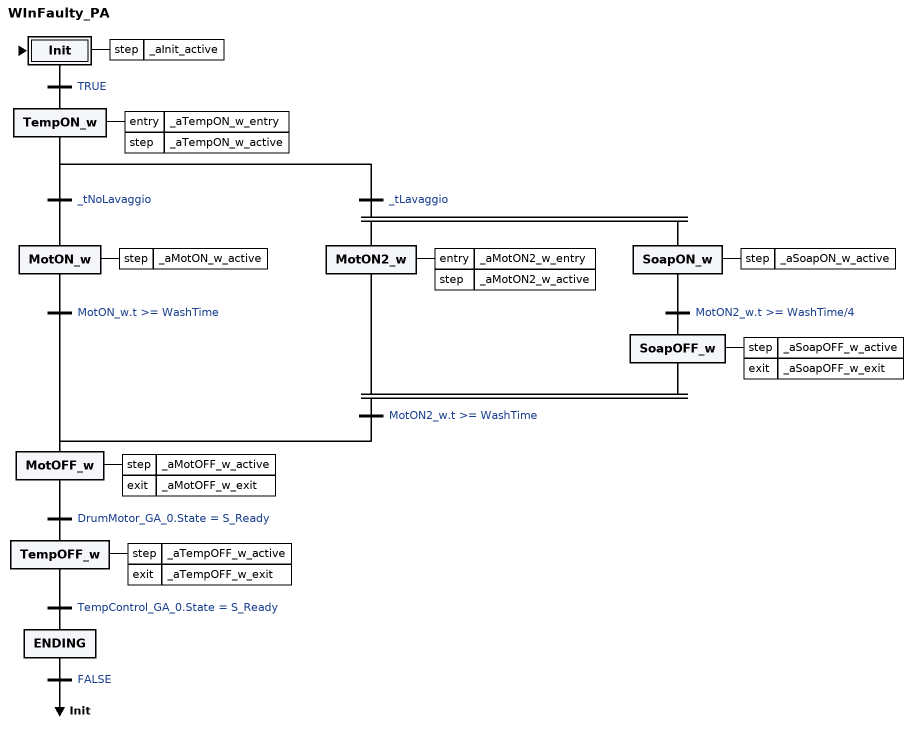
INITIAL_STEP Init:
    _aInit_active(N);  // step action
END_STEP
TRANSITION FROM Init TO TempON_w
    := TRUE;
END_TRANSITION
STEP TempON_w:
    _aTempON_w_entry(P1);  // entry action
    _aTempON_w_active(N);  // step action
END_STEP
TRANSITION FROM TempON_w TO MotON_w
    := _tNoLavaggio;
END_TRANSITION
STEP MotON_w:
    _aMotON_w_active(N);  // step action
END_STEP
TRANSITION FROM MotON_w TO MotOFF_w
    := MotON_w.t >= WashTime;
END_TRANSITION
TRANSITION FROM TempON_w TO (MotON2_w, SoapON_w)
    := _tLavaggio;
END_TRANSITION
STEP MotON2_w:
    _aMotON2_w_entry(P1);  // entry action
    _aMotON2_w_active(N);  // step action
END_STEP
STEP SoapON_w:
    _aSoapON_w_active(N);  // step action
END_STEP
TRANSITION FROM SoapON_w TO SoapOFF_w
    := MotON2_w.t >= WashTime/4;
END_TRANSITION
STEP SoapOFF_w:
    _aSoapOFF_w_active(N);  // step action
    _aSoapOFF_w_exit(P0);  // exit action
END_STEP
TRANSITION FROM (MotON2_w, SoapOFF_w) TO MotOFF_w
    := MotON2_w.t >= WashTime;
END_TRANSITION
STEP MotOFF_w:
    _aMotOFF_w_active(N);  // step action
    _aMotOFF_w_exit(P0);  // exit action
END_STEP
TRANSITION FROM MotOFF_w TO TempOFF_w
    := DrumMotor_GA_0.State = S_Ready;
END_TRANSITION
STEP TempOFF_w:
    _aTempOFF_w_active(N);  // step action
    _aTempOFF_w_exit(P0);  // exit action
END_STEP
TRANSITION FROM TempOFF_w TO ENDING
    := TempControl_GA_0.State = S_Ready;
END_TRANSITION
STEP ENDING:
END_STEP
TRANSITION FROM ENDING TO Init
    := FALSE;
END_TRANSITION

ACTION _aTempRegON_exit:

END_ACTION

ACTION _aTempOFF_w_active:
TempControl_GA_0.StopTemp := TRUE;
TempControl_GA_0.StartTemp := FALSE;
END_ACTION

ACTION _aInit_active:

END_ACTION

ACTION _aMotON_w_active:
IF DrumMotor_GA_0.State = S_Ready THEN
	DrumMotor_GA_0.StartMotor := TRUE;
END_IF
END_ACTION

ACTION _aTempOFF_w_exit:
TempControl_GA_0.StopTemp := FALSE;
IDOL := TRUE;
//Idol := TRUE;
END_ACTION

TRANSITION _tLavaggio:
(TempControl_GA_0.TempOk OR TempControl_GA_0.failure = Heat) AND Washing_P = Lavaggio AND WaterManagement_GA_0.flt_case = late
END_TRANSITION

ACTION _aStartMotor2_active:
IF DrumMotor_GA_0.State = S_Ready THEN
	DrumMotor_GA_0.StartMotor := TRUE;
END_IF
END_ACTION

ACTION _aTempON_w_active:

IF TempControl_GA_0.State = S_Ready AND TempControl_GA_0.failure = None THEN
	TempControl_GA_0.StartTemp := TRUE;
END_IF
END_ACTION

ACTION _aMotOFF_w_exit:
DrumMotor_GA_0.StopMotor := FALSE;
END_ACTION

ACTION _aTempON_w_entry:

IF WaterManagement_GA_0.flt_case = mid THEN
(*esecuzione degradata più lunga della fase in cui mi trovo con temperatura fissata a 30 gradi per sicurezza*)
	TempControl_GA_0.StartWhat := Warm30;
	WashTime:= T#10S;
ELSIF WaterManagement_GA_0.flt_case = late THEN
	TempControl_GA_0.StartWhat := SelectedTemp;
END_IF
END_ACTION

ACTION _aMotON2_w_entry:
WashTime:= T#10S;
END_ACTION

TRANSITION _tNoLavaggio:
(TempControl_GA_0.TempOk OR TempControl_GA_0.failure = Heat)AND (Washing_P <> Lavaggio OR WaterManagement_GA_0.flt_case = mid)
END_TRANSITION

ACTION _aSoapOFF_w_exit:
SoapEmptying_GA_0.StopSoap := FALSE;
END_ACTION

ACTION _aMotON2_w_active:

IF DrumMotor_GA_0.State = S_Ready THEN
	DrumMotor_GA_0.StartMotor := TRUE;
END_IF
END_ACTION

ACTION _aSoapON_w_active:
IF SoapEmptying_GA_0.State = S_Ready THEN
	SoapEmptying_GA_0.StartSoap := TRUE;
END_IF
END_ACTION

ACTION _aSoapOFF_w_active:
SoapEmptying_GA_0.StopSoap := TRUE;
SoapEmptying_GA_0.StartSoap := FALSE;
END_ACTION

ACTION _aMotOFF_w_active:
DrumMotor_GA_0.StopMotor := TRUE;
DrumMotor_GA_0.StartMotor := FALSE;
END_ACTION

END_PROGRAM

// Device/Application/PROGRAMs/Policy_Automatas/Child_PAs/FaultManagerPAs/HeatFaulty_PA
PROGRAM HeatFaulty_PA
VAR
END_VAR
VAR_INPUT
	SFCInit:BOOL;
	SFCPause: BOOL;
END_VAR

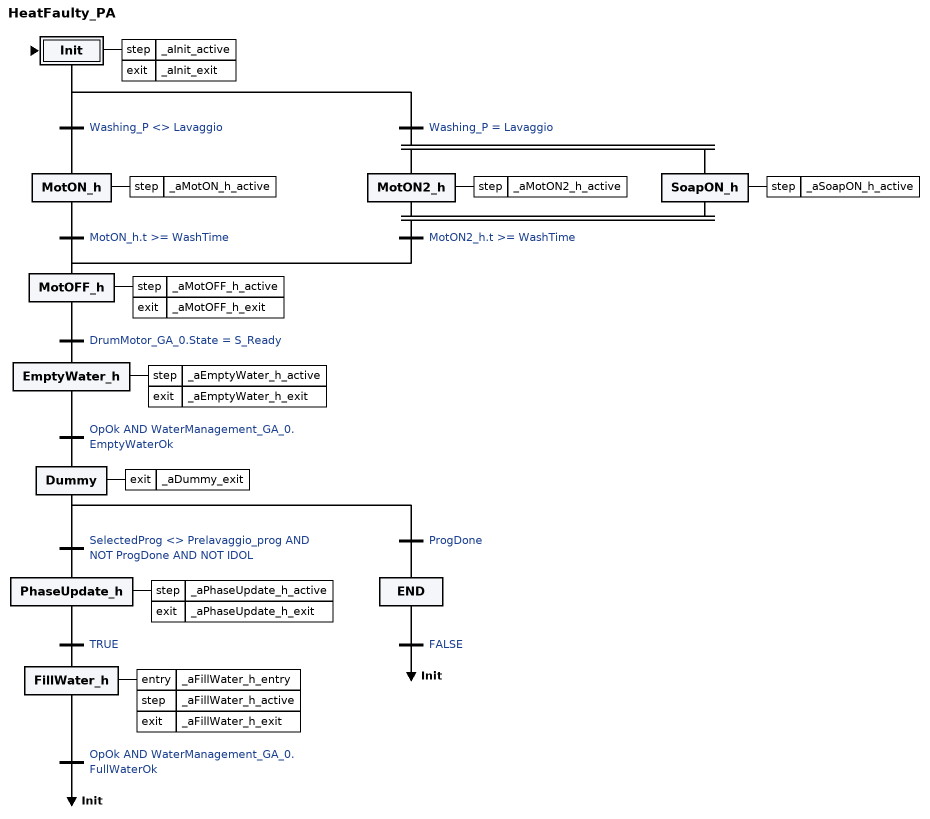
INITIAL_STEP Init:
    _aInit_active(N);  // step action
    _aInit_exit(P0);  // exit action
END_STEP
TRANSITION FROM Init TO MotON_h
    := Washing_P <> Lavaggio;
END_TRANSITION
STEP MotON_h:
    _aMotON_h_active(N);  // step action
END_STEP
TRANSITION FROM MotON_h TO MotOFF_h
    := MotON_h.t >= WashTime;
END_TRANSITION
TRANSITION FROM Init TO (MotON2_h, SoapON_h)
    := Washing_P = Lavaggio;
END_TRANSITION
STEP MotON2_h:
    _aMotON2_h_active(N);  // step action
END_STEP
STEP SoapON_h:
    _aSoapON_h_active(N);  // step action
END_STEP
TRANSITION FROM (MotON2_h, SoapON_h) TO MotOFF_h
    := MotON2_h.t >= WashTime;
END_TRANSITION
STEP MotOFF_h:
    _aMotOFF_h_active(N);  // step action
    _aMotOFF_h_exit(P0);  // exit action
END_STEP
TRANSITION FROM MotOFF_h TO EmptyWater_h
    := DrumMotor_GA_0.State = S_Ready;
END_TRANSITION
STEP EmptyWater_h:
    _aEmptyWater_h_active(N);  // step action
    _aEmptyWater_h_exit(P0);  // exit action
END_STEP
TRANSITION FROM EmptyWater_h TO Dummy
    := OpOk AND WaterManagement_GA_0.EmptyWaterOk;
END_TRANSITION
STEP Dummy:
    _aDummy_exit(P0);  // exit action
END_STEP
TRANSITION FROM Dummy TO PhaseUpdate_h
    := SelectedProg <> Prelavaggio_prog AND NOT ProgDone AND NOT IDOL;
END_TRANSITION
TRANSITION FROM Dummy TO END
    := ProgDone;
END_TRANSITION
STEP END:
END_STEP
TRANSITION FROM END TO Init
    := FALSE;
END_TRANSITION
STEP PhaseUpdate_h:
    _aPhaseUpdate_h_active(N);  // step action
    _aPhaseUpdate_h_exit(P0);  // exit action
END_STEP
TRANSITION FROM PhaseUpdate_h TO FillWater_h
    := TRUE;
END_TRANSITION
STEP FillWater_h:
    _aFillWater_h_entry(P1);  // entry action
    _aFillWater_h_active(N);  // step action
    _aFillWater_h_exit(P0);  // exit action
END_STEP
TRANSITION FROM FillWater_h TO Init
    := OpOk AND WaterManagement_GA_0.FullWaterOk;
END_TRANSITION

ACTION _aDummy_exit:
IF ProgDone OR WaterManagement_GA_0.failure = WaterIn THEN 
	IDOL := TRUE;
	SetBools(2,FALSE); //spegnimento di tutti i led per le fasi HMI
	ProgDone := FALSE;
END_IF
END_ACTION

ACTION _aFillWater_h_active:
CASE Action_S OF //macchina a stati implementata con uno switch case, funziona grazie al modello di esecuzione con while intrinseco
//n.b. per fare la diagnostica di alto livello di tipo A tra politica e GA dovrei aggiungere un else nell'if per il caso il cui non si ver
//verifica mai lo stato ready(anomalia)
Start_Action: IF WaterManagement_GA_0.State = S_Ready THEN 
				 WaterManagement_GA_0.Do_ := TRUE;
				 WaterManagement_GA_0.DoWhat := Do_WaterFilling;
				 Action_S := Wait_Compl;
			  END_IF
			  
Wait_Compl: IF WaterManagement_GA_0.Done AND WaterManagement_GA_0.State = S_Busy THEN 
			   WaterManagement_GA_0.Do_ := FALSE;
			   Action_S := SetOpOk;
			ELSIF NOT WaterManagement_GA_0.Done AND WaterManagement_GA_0.State = S_Fault THEN 
				WaterManagement_GA_0.Do_ := FALSE;
				Action_S := Start_Action;
			END_IF
//protocollo di handshake di set reset del do e done da parte di politica e ga per evitare attivazioni multiple
SetOpOk: IF NOT WaterManagement_GA_0.Done THEN
			OpOk := TRUE;
	     END_IF
END_CASE
END_ACTION

ACTION _aMotON_h_active:
IF DrumMotor_GA_0.State = S_Ready THEN
	DrumMotor_GA_0.StartMotor := TRUE;
END_IF
END_ACTION

ACTION _aMotON2_h_active:
IF DrumMotor_GA_0.State = S_Ready THEN
	DrumMotor_GA_0.StartMotor := TRUE;
END_IF
END_ACTION

ACTION _aInit_exit:

END_ACTION

ACTION _aEmptyWater_h_exit:
OpOk := FALSE;
Action_S := Start_Action;
END_ACTION

ACTION _aMotOFF_h_exit:
DrumMotor_GA_0.StopMotor := FALSE;
SoapEmptying_GA_0.StopSoap := FALSE;
END_ACTION

ACTION _aPhaseUpdate_h_active:
IF SelectedProg = LavaggioCompleto_prog THEN
	CASE Washing_P OF 
	Prelavaggio: Washing_P := Lavaggio;
	
	Lavaggio : Washing_P := Risciacquo;
			   ProgDone := TRUE;
	END_CASE
END_IF

IF SelectedProg = Lavaggio_prog AND Washing_P = Lavaggio THEN
	Washing_P := Risciacquo;
	ProgDone := TRUE;
END_IF
END_ACTION

ACTION _aSoapON_h_active:
IF SoapEmptying_GA_0.State = S_Ready THEN
	SoapEmptying_GA_0.StartSoap := TRUE;
END_IF
END_ACTION

ACTION _aEmptyWater_h_active:
CASE Action_S OF //macchina a stati implementata con uno switch case, funziona grazie al modello di esecuzione con while intrinseco
//n.b. per fare la diagnostica di alto livello di tipo A tra politica e GA dovrei aggiungere un else nell'if per il caso il cui non si ver
//verifica mai lo stato ready(anomalia)
Start_Action: IF WaterManagement_GA_0.State = S_Ready THEN 
				 WaterManagement_GA_0.Do_ := TRUE;
				 WaterManagement_GA_0.DoWhat := Do_WaterEmptying;
				 Action_S := Wait_Compl;
			  END_IF
			  
Wait_Compl: IF WaterManagement_GA_0.Done AND WaterManagement_GA_0.State = S_Busy THEN 
			   WaterManagement_GA_0.Do_ := FALSE;
			   Action_S := SetOpOk;
			ELSIF NOT WaterManagement_GA_0.Done AND WaterManagement_GA_0.State = S_Fault THEN 
				WaterManagement_GA_0.Do_ := FALSE;
				Action_S := Start_Action;
			END_IF
//protocollo di handshake di set reset del do e done da parte di politica e ga per evitare attivazioni multiple
SetOpOk: IF NOT WaterManagement_GA_0.Done THEN
			OpOk := TRUE;
	     END_IF
END_CASE
END_ACTION

ACTION _aPhaseUpdate_h_exit:
prewash := FALSE;
wash := FALSE;
rinse := FALSE;
END_ACTION

ACTION _aFillWater_h_entry:

	CASE Washing_P OF 
	Prelavaggio: prewash := TRUE;
	Lavaggio: wash := TRUE;
	Risciacquo: rinse := TRUE;
	END_CASE
END_ACTION

ACTION _aInit_active:

END_ACTION

ACTION _aMotOFF_h_active:
DrumMotor_GA_0.StopMotor := TRUE;
DrumMotor_GA_0.StartMotor := FALSE;

SoapEmptying_GA_0.StopSoap := TRUE;
SoapEmptying_GA_0.StartSoap := FALSE;
END_ACTION

ACTION _aFillWater_h_exit:
OpOk := FALSE;
Action_S := Start_Action;
END_ACTION

END_PROGRAM

// Device/Application/FUNCTIONs/FaultHMI
FUNCTION FaultHMI : BOOL
VAR_INPUT
	Fault : FaultType;
	value : BOOL;
END_VAR
VAR
END_VAR

CASE Fault OF
	WaterIn: water_in_alarm := value;
	WaterOut: water_out_alarm := value;
	Heat: heat_alarm := value;
END_CASE

END_FUNCTION

// Device/Application/FUNCTIONs/CheckFault
FUNCTION CheckFault : FaultType
VAR_INPUT
END_VAR
VAR
END_VAR

IF WaterManagement_GA_0.State = S_Fault THEN
	CheckFault := WaterManagement_GA_0.failure;
ELSIF TempControl_GA_0.State = S_Fault THEN
	CheckFault := heat;
ELSE 
	CheckFault := None;
END_IF

END_FUNCTION

// Device/Application/PROGRAMs/Simulation_Program
PROGRAM Simulation_Program
VAR
		bulls_eye_open_past	:BOOL := TRUE;
END_VAR

(*Temperature value simulation*)
IF ((GVL.hot)AND(NOT GVL.heat_fail)) THEN 
	GVL.temperature := GVL.temperature + 1;
ELSE
	GVL.temperature := GVL.temperature - 1;
END_IF

IF GVL.temperature > 100 THEN 
	GVL.temperature := 100;
END_IF

IF GVL.temperature < 0 THEN 
	GVL.temperature := 0;
END_IF


(*Soap level simulation*)
IF GVL.fillsoap THEN 
	GVL.soaplevel := GVL.soaplevel + 5;
ELSIF GVL.emptysoap THEN 
	GVL.soaplevel := GVL.soaplevel - 3;
END_IF

IF GVL.soaplevel >= 50 THEN 
	GVL.soaplevel := 50;
	GVL.fillsoap := FALSE;
END_IF

IF GVL.soaplevel < 0 THEN 
	GVL.soaplevel := 0;
END_IF


(*Door state simulation*)
IF ((GVL.bulls_eye_open <> bulls_eye_open_past)AND(NOT GVL.bulls_eye_lock)) THEN 
	bulls_eye_open_past := GVL.bulls_eye_open ;
ELSIF GVL.bulls_eye_lock THEN
	GVL.bulls_eye_open := bulls_eye_open_past;
END_IF


(*Water level simulation*)
IF ((GVL.fillwater)AND(NOT GVL.water_in_fail)) THEN 
	GVL.waterlevel := GVL.waterlevel + 2;
ELSIF ((GVL.emptywater)AND(NOT GVL.water_out_fail)) THEN
	GVL.waterlevel := GVL.waterlevel - 4;
END_IF

IF GVL.waterlevel > 150 THEN 
	GVL.waterlevel := 150;
END_IF

IF GVL.waterlevel < 0 THEN 
	GVL.waterlevel := 0;
END_IF


(*Motor simulation*)
IF (GVL.motor_on) THEN 
	GVL.motor := GVL.motor + 10;
END_IF

IF GVL.motor > 360 THEN 
	GVL.motor := 0;
END_IF

END_PROGRAM

// Device/Application/PROGRAMs/GA_Collector
PROGRAM GA_Collector
VAR
END_VAR

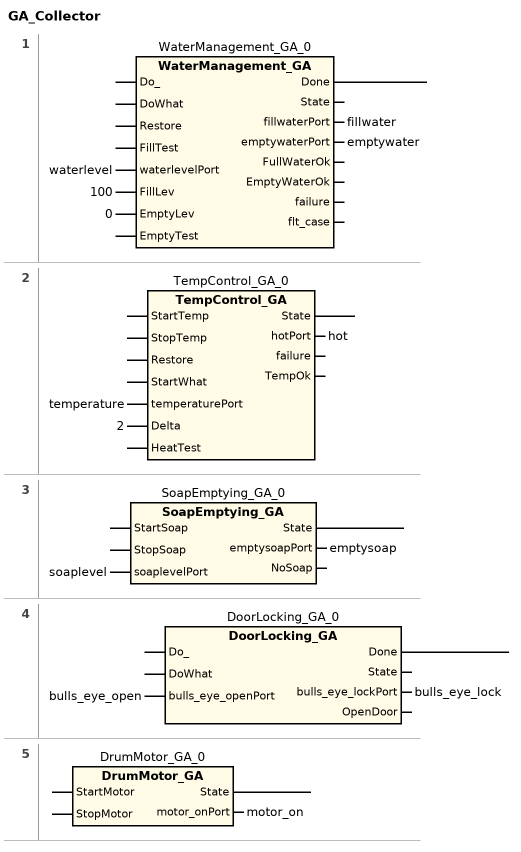
// NETWORK 1
WaterManagement_GA_0(
    waterlevelPort := waterlevel,
    FillLev := 100,
    EmptyLev := 0,
    fillwaterPort => fillwater,
    emptywaterPort => emptywater); // WaterManagement_GA

// NETWORK 2
TempControl_GA_0(temperaturePort := temperature, Delta := 2, hotPort => hot); // TempControl_GA

// NETWORK 3
SoapEmptying_GA_0(soaplevelPort := soaplevel, emptysoapPort => emptysoap); // SoapEmptying_GA

// NETWORK 4
DoorLocking_GA_0(bulls_eye_openPort := bulls_eye_open, bulls_eye_lockPort => bulls_eye_lock); // DoorLocking_GA

// NETWORK 5
DrumMotor_GA_0(motor_onPort => motor_on); // DrumMotor_GA

END_PROGRAM

// Device/Application/FUNCTIONBLOCKs/GAs/WaterManagement_GA
FUNCTION_BLOCK WaterManagement_GA
VAR_INPUT
	Do_: BOOL;
	DoWhat: WaterDoWhats;
	Restore: BOOL;
	FillTest: BOOL;
	waterlevelPort: INT;
	FillLev: INT;
	EmptyLev: INT;
	EmptyTest: BOOL;
END_VAR
VAR_OUTPUT
	Done: BOOL;
	State: STATE_FB;
	fillwaterPort: BOOL;
	emptywaterPort: BOOL;
	FullWaterOk: BOOL;
	EmptyWaterOk: BOOL;
	failure: FaultType;
	flt_case : WinFlt_cases;
END_VAR
VAR
	LevStore: INT;
END_VAR

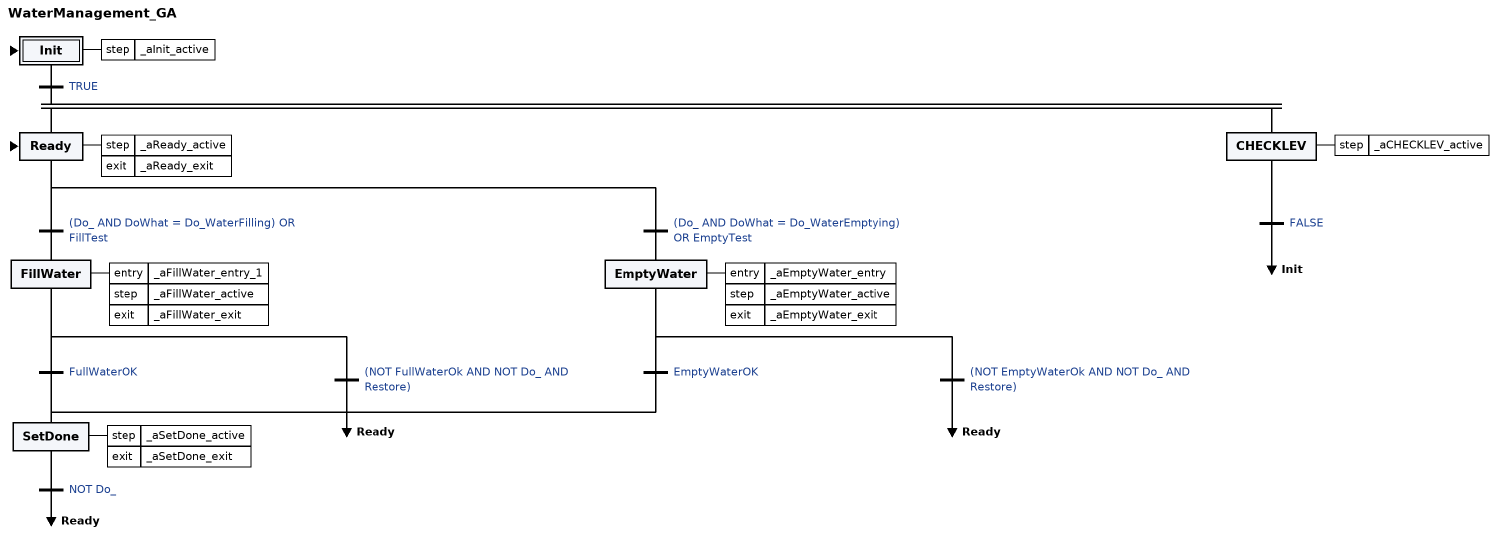
INITIAL_STEP Init:
    _aInit_active(N);  // step action
END_STEP
TRANSITION FROM Init TO (Ready, CHECKLEV)
    := TRUE;
END_TRANSITION
STEP Ready:
    _aReady_active(N);  // step action
    _aReady_exit(P0);  // exit action
END_STEP
STEP CHECKLEV:
    _aCHECKLEV_active(N);  // step action
END_STEP
TRANSITION FROM CHECKLEV TO Init
    := FALSE;
END_TRANSITION
TRANSITION FROM Ready TO FillWater
    := (Do_ AND DoWhat = Do_WaterFilling) OR FillTest;
END_TRANSITION
STEP FillWater:
    _aFillWater_entry_1(P1);  // entry action
    _aFillWater_active(N);  // step action
    _aFillWater_exit(P0);  // exit action
END_STEP
TRANSITION FROM FillWater TO SetDone
    := FullWaterOK;
END_TRANSITION
TRANSITION FROM FillWater TO Ready
    := (NOT FullWaterOk AND NOT Do_ AND Restore);
END_TRANSITION
TRANSITION FROM Ready TO EmptyWater
    := (Do_ AND DoWhat = Do_WaterEmptying) OR EmptyTest;
END_TRANSITION
STEP EmptyWater:
    _aEmptyWater_entry(P1);  // entry action
    _aEmptyWater_active(N);  // step action
    _aEmptyWater_exit(P0);  // exit action
END_STEP
TRANSITION FROM EmptyWater TO SetDone
    := EmptyWaterOK;
END_TRANSITION
TRANSITION FROM EmptyWater TO Ready
    := (NOT EmptyWaterOk AND NOT Do_ AND Restore);
END_TRANSITION
STEP SetDone:
    _aSetDone_active(N);  // step action
    _aSetDone_exit(P0);  // exit action
END_STEP
TRANSITION FROM SetDone TO Ready
    := NOT Do_;
END_TRANSITION

ACTION _aSetDone_exit:
Done := FALSE;
END_ACTION

ACTION _aEmptyWater_exit:
emptywaterPort := FALSE;
END_ACTION

ACTION _aFillWater_exit:
fillwaterPort := FALSE;
PolicyEval := HealthyPA;
END_ACTION

ACTION _aInit_active:
State := S_Init;
failure := None;
END_ACTION

ACTION _aEmptyWater_active:
emptywaterPort := TRUE;

(*Diagnostica di basso livello di corretto comportamento di attuatori e sensori, incapsulata interna al GA per verificare la presenza di anomalia relativa ad otturazione del tubo
di scarico dell'acqua dalla lavatrice*)
//FAULT DETECTION
IF LevStore <=  waterlevelPort AND NOT EmptyTest THEN
	State := S_Fault;
	failure := WaterOut;
	PolicyEval := KilledPA;
	emptywaterPort := FALSE; (*QUESTA è GIà UNA PRIMA FORMA DI GESTIONE DEL FAULT INTERNA AL GA*)
ELSE LevStore :=  waterlevelPort;
END_IF

IF Do_Abort THEN
	emptywaterPort := FALSE;
	LevStore :=  waterlevelPort+1;
END_IF
END_ACTION

ACTION _aReady_exit:
State := S_Busy;
END_ACTION

ACTION _aReady_active:
State := S_Ready;
END_ACTION

ACTION _aCHECKLEV_active:
IF waterlevelPort >= FillLev THEN
	FullWaterOk := TRUE;
	ELSE
	FullWaterOk := FALSE;
END_IF

IF waterlevelPort <= EmptyLev THEN
	EmptyWaterOk := TRUE;
	ELSE
	EmptyWaterOk := FALSE;
END_IF
END_ACTION

ACTION _aEmptyWater_entry:
LevStore :=  waterlevelPort+1;
END_ACTION

ACTION _aSetDone_active:
Done := TRUE;
END_ACTION

ACTION _aFillWater_active:
fillwaterPort := TRUE;


(*Diagnostica di basso livello di corretto comportamento di attuatori e sensori, incapsulata interna al GA per verificare la presenza di anomalia relativa ad otturazione del tubo
di immissione dell'acqua nella lavatrice*)
//FAULT DETECTION
IF LevStore >=  waterlevelPort AND fillwaterPort AND NOT FillTest THEN
	State := S_Fault;
	failure := WaterIn;
	fillwaterPort := FALSE; (*QUESTA è GIà UNA PRIMA FORMA DI GESTIONE DEL FAULT INTERNA AL GA*)
	
	//FAULT ISOLATION CHECK
	IF waterlevelPort < 20 THEN
		PolicyEval := KilledPA;
		flt_case := early;
	ELSE
		PolicyEval := FaultyPA;
			IF waterlevelPort >=20 AND waterlevelPort < 70 THEN
				flt_case := mid;
			ELSE 
				flt_case := late;
			END_IF
	END_IF
	
ELSE LevStore :=  waterlevelPort;
END_IF

//PAUSA QUANDO SPENGO IL PULSANTE DI RUN DURANTE L'ESECUZIONE DI UN PROGRAMMA
IF Do_Abort THEN 
	fillwaterPort := FALSE;
	LevStore := waterlevelPort - 1; //necessario per evitare il fault se premo il pulsante di stop durante il riempimento
END_IF
END_ACTION

ACTION _aFillWater_entry_1:
LevStore := waterlevelPort - 1; //altrimenti entrerebbe in fault subito quando ancora deve riempire l'acqua
END_ACTION

END_FUNCTION_BLOCK

// Device/Application/FUNCTIONBLOCKs/GAs/TempControl_GA
FUNCTION_BLOCK TempControl_GA
VAR_INPUT
	StartTemp: BOOL;
	StopTemp: BOOL;
	Restore: BOOL;
	StartWhat: WMTemps;	
//StartWhat: TempStartWhats;
	temperaturePort: INT;
	Delta: INT;
	HeatTest: BOOL;

END_VAR
VAR_OUTPUT
	State: STATE_FB;
	hotPort: BOOL;
	TempOk: BOOL;
	failure: FaultType;
	
END_VAR
VAR
	TempStore: INT;
END_VAR

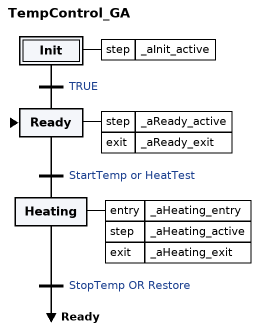
INITIAL_STEP Init:
    _aInit_active(N);  // step action
END_STEP
TRANSITION FROM Init TO Ready
    := TRUE;
END_TRANSITION
STEP Ready:
    _aReady_active(N);  // step action
    _aReady_exit(P0);  // exit action
END_STEP
TRANSITION FROM Ready TO Heating
    := StartTemp or HeatTest;
END_TRANSITION
STEP Heating:
    _aHeating_entry(P1);  // entry action
    _aHeating_active(N);  // step action
    _aHeating_exit(P0);  // exit action
END_STEP
TRANSITION FROM Heating TO Ready
    := StopTemp OR Restore;
END_TRANSITION

ACTION _aReady_exit:
State := S_Busy;
END_ACTION

ACTION _aInit_active:
State := S_Init;
failure := None;
END_ACTION

ACTION _aReady_active:
State := S_Ready;
END_ACTION

ACTION _aHeating_entry:
TempStore := temperaturePort-1;
END_ACTION

ACTION _aHeating_exit:
hotPort := FALSE;
PolicyEval := HealthyPA;
END_ACTION

ACTION _aHeating_active:
(*Diagnostica di basso livello di corretto comportamento di attuatori e sensori, incapsulata interna al GA per verificare la presenza di anomalia relativa 
a rottura di resistenza di riscaldamento dell'acqua lavatrice*)

//FAULT DETECTION 
IF hotPort AND TempStore >=  temperaturePort THEN
	State := S_Fault;
	failure := Heat;
	hotPort := FALSE; (*QUESTA è GIà UNA PRIMA FORMA DI GESTIONE DEL FAULT INTERNA AL GA*)
	PolicyEval := FaultyPA;
ELSE TempStore :=  temperaturePort;
	IF temperaturePort < StartWhat - Delta THEN
		hotPort := TRUE;
		tempOK := FALSE;
	ELSIF temperaturePort > StartWhat + Delta THEN
		hotPort := FALSE;
		tempOK := FALSE;
	ELSE
		tempOK := TRUE;
	END_IF
END_IF

//PAUSA DELL'ESECUZIONE SE SPENGO IL PULSANTE DI RUN DURANTE L'ESECUZIONE
IF Do_Abort THEN
	hotPort := FALSE;
END_IF
END_ACTION

END_FUNCTION_BLOCK

// Device/Application/FUNCTIONBLOCKs/GAs/SoapEmptying_GA
FUNCTION_BLOCK SoapEmptying_GA
VAR_INPUT
	StartSoap: BOOL;
	StopSoap: BOOL;
	soaplevelPort: INT;
END_VAR
VAR_OUTPUT
	State: STATE_FB;
	emptysoapPort: BOOL;
	NoSoap: BOOL;
END_VAR
VAR
END_VAR

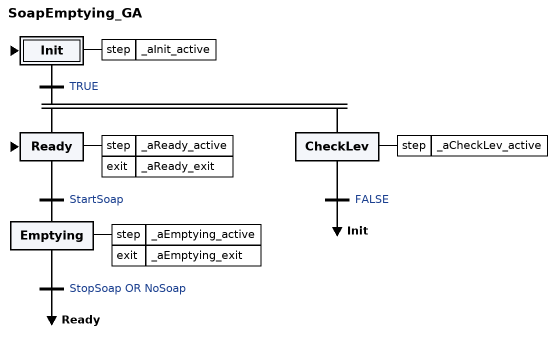
INITIAL_STEP Init:
    _aInit_active(N);  // step action
END_STEP
TRANSITION FROM Init TO (Ready, CheckLev)
    := TRUE;
END_TRANSITION
STEP Ready:
    _aReady_active(N);  // step action
    _aReady_exit(P0);  // exit action
END_STEP
STEP CheckLev:
    _aCheckLev_active(N);  // step action
END_STEP
TRANSITION FROM CheckLev TO Init
    := FALSE;
END_TRANSITION
TRANSITION FROM Ready TO Emptying
    := StartSoap;
END_TRANSITION
STEP Emptying:
    _aEmptying_active(N);  // step action
    _aEmptying_exit(P0);  // exit action
END_STEP
TRANSITION FROM Emptying TO Ready
    := StopSoap OR NoSoap;
END_TRANSITION

ACTION _aReady_active:
State := S_Ready;
END_ACTION

ACTION _aCheckLev_active:
IF soaplevelPort > 0 THEN
	NoSoap := FALSE;
ELSE
	NoSoap := TRUE;
END_IF
END_ACTION

ACTION _aReady_exit:
State := S_Busy;
END_ACTION

ACTION _aInit_active:
State := S_Init;
END_ACTION

ACTION _aEmptying_active:
emptySoapPort := TRUE;
IF Do_Abort THEN
	emptySoapPort := FALSE;
END_IF
END_ACTION

ACTION _aEmptying_exit:
emptySoapPort := FALSE;
END_ACTION

END_FUNCTION_BLOCK

// Device/Application/FUNCTIONBLOCKs/GAs/DoorLocking_GA
FUNCTION_BLOCK DoorLocking_GA
VAR_INPUT
	Do_ : BOOL;
	DoWhat : LockerDoWhats;
	bulls_eye_openPort : BOOL;
END_VAR
VAR_OUTPUT
	Done: BOOL;
	State: STATE_FB;
	bulls_eye_lockPort: BOOL;

	OpenDoor: BOOL;
END_VAR
VAR
END_VAR

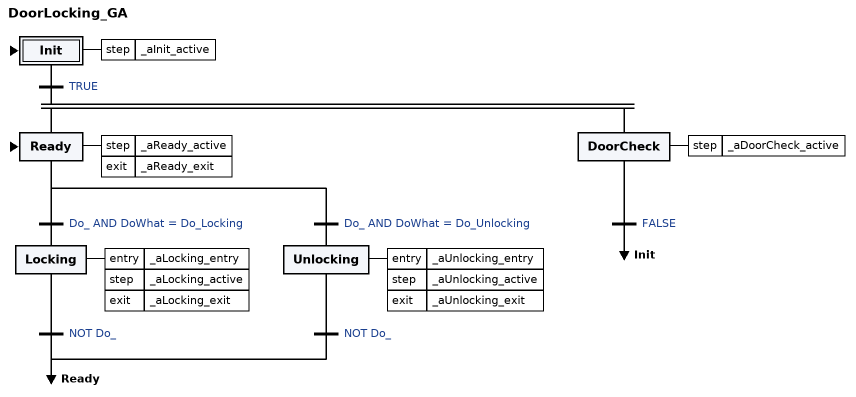
INITIAL_STEP Init:
    _aInit_active(N);  // step action
END_STEP
TRANSITION FROM Init TO (Ready, DoorCheck)
    := TRUE;
END_TRANSITION
STEP Ready:
    _aReady_active(N);  // step action
    _aReady_exit(P0);  // exit action
END_STEP
STEP DoorCheck:
    _aDoorCheck_active(N);  // step action
END_STEP
TRANSITION FROM DoorCheck TO Init
    := FALSE;
END_TRANSITION
TRANSITION FROM Ready TO Locking
    := Do_ AND DoWhat = Do_Locking;
END_TRANSITION
STEP Locking:
    _aLocking_entry(P1);  // entry action
    _aLocking_active(N);  // step action
    _aLocking_exit(P0);  // exit action
END_STEP
TRANSITION FROM Locking TO Ready
    := NOT Do_;
END_TRANSITION
TRANSITION FROM Ready TO Unlocking
    := Do_ AND DoWhat = Do_Unlocking;
END_TRANSITION
STEP Unlocking:
    _aUnlocking_entry(P1);  // entry action
    _aUnlocking_active(N);  // step action
    _aUnlocking_exit(P0);  // exit action
END_STEP
TRANSITION FROM Unlocking TO Ready
    := NOT Do_;
END_TRANSITION

ACTION _aLocking_active:
Done := TRUE;
END_ACTION

ACTION _aReady_active:
State := S_Ready;
END_ACTION

ACTION _aInit_active:
State := S_init;
END_ACTION

ACTION _aUnlocking_active:
Done := TRUE;
END_ACTION

ACTION _aReady_exit:
State := S_Busy;
END_ACTION

ACTION _aLocking_entry:
bulls_eye_lockPort := TRUE;
END_ACTION

ACTION _aUnlocking_entry:
bulls_eye_lockPort := FALSE;
END_ACTION

ACTION _aUnlocking_exit:
Done := FALSE;
END_ACTION

ACTION _aLocking_exit:
Done := FALSE;
END_ACTION

ACTION _aDoorCheck_active:
OpenDoor := bulls_eye_openPort;
END_ACTION

END_FUNCTION_BLOCK

// Device/Application/FUNCTIONBLOCKs/GAs/DrumMotor_GA
FUNCTION_BLOCK DrumMotor_GA
VAR_INPUT
	StartMotor: BOOL;
	StopMotor: BOOL;
END_VAR
VAR_OUTPUT
	State: STATE_FB;
	motor_onPort: BOOL;
END_VAR
VAR
END_VAR

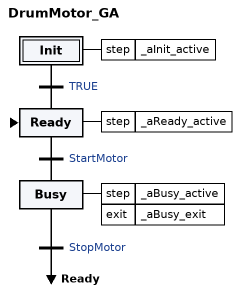
INITIAL_STEP Init:
    _aInit_active(N);  // step action
END_STEP
TRANSITION FROM Init TO Ready
    := TRUE;
END_TRANSITION
STEP Ready:
    _aReady_active(N);  // step action
END_STEP
TRANSITION FROM Ready TO Busy
    := StartMotor;
END_TRANSITION
STEP Busy:
    _aBusy_active(N);  // step action
    _aBusy_exit(P0);  // exit action
END_STEP
TRANSITION FROM Busy TO Ready
    := StopMotor;
END_TRANSITION

ACTION _aBusy_active:
State := S_Busy;
motor_onPort := TRUE;
IF Do_Abort THEN
	motor_onPort := FALSE;
END_IF
END_ACTION

ACTION _aReady_active:
State := S_Ready;
END_ACTION

ACTION _aInit_active:
State := S_Init;
END_ACTION

ACTION _aBusy_exit:
motor_onPort := FALSE;
END_ACTION

END_FUNCTION_BLOCK

// Device/Application/Visualization
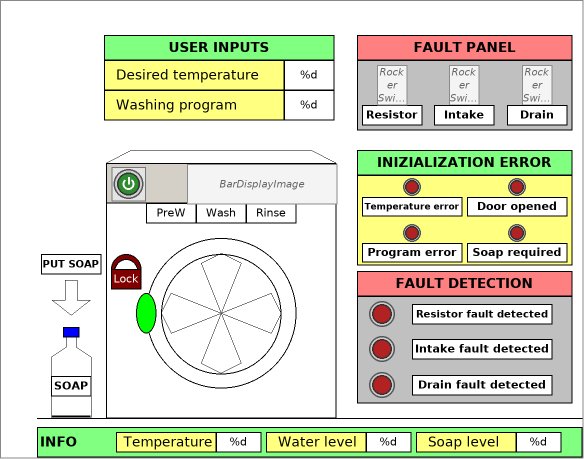
VISUALIZATION Visualization  // 584x459
    Line (37,418) (582,418)
    Rectangle (106,178 230x240)
    Ellipse (162,254 118x118)
    Rectangle (161,255 120x120)
        p1126004900: -GVL.waterlevel/3*2
    Ellipse (146,238 150x150)
    Ellipse (161,254 120x120)
    Polygon (221,253) (201,263) (221,313) (171,293) (161,313) (171,333) (221,313) (201,363) (221,373) (241,363) (221,313) (271,333) (281,313) (271,293) (221,313) (241,263)
        p2858320360: GVL.motor
    Ellipse (136,293 20x40), colour toggle: GVL.bulls_eye_open
        toggle GVL.bulls_eye_open
    Ellipse (111,254 30x30), colour toggle: GVL.bulls_eye_lock
    Ellipse (114,259 24x27)
    Rectangle (111,269 30x20), "Lock", colour toggle: GVL.bulls_eye_lock
    Rectangle (106,163 230x40)
    Rectangle (146,203 50x20), "PreW", colour toggle: GVL.prewash
    Rectangle (196,203 50x20), "Wash", colour toggle: GVL.wash
    Rectangle (246,203 50x20), "Rinse", colour toggle: GVL.rinse
    Polygon (106,163) (131,150) (311,150) (336,163)
    PowerSwitch (111,167 35x34), variable: GVL.run, behaviour: TOGGLE, style: Switch-PowerSwitch-Green
    BarDisplayImage (187,164 150x40), value: GVL.temperature, style: BarDisplayImage-Gray, scale format: %.0f, scale 0..90
    Polygon (51,417) (51,357) (66,347) (66,332) (76,332) (76,347) (91,357) (91,417)
    Rectangle (63,327 16x10)
    Rectangle (104,60 180x30), "Desired temperature"
        OnMouseDown: write GVL.temp_number via VisuDialogs.Numpad, min 0, max 100, format 0
    Rectangle (104,90 180x30), "Washing program"
        OnMouseDown: write GVL.prog_number via VisuDialogs.Numpad, min 0, max 100, format 0
    Rectangle (104,35 230x25), "USER INPUTS"
    Rectangle (284,60 50x30), "%d", text variable: GVL.temp_number
    Rectangle (284,90 50x30), "%d", text variable: GVL.prog_number
    Rectangle (37,427 545x30), "INFO"
    Rectangle (116,432 100x20), "Temperature"
    Rectangle (357,150 215x25), "INIZIALIZATION ERROR"
    Rectangle (216,432 45x20), "%d", text variable: GVL.temperature
    Rectangle (266,432 100x20), "Water level"
    Rectangle (366,432 45x20), "%d", text variable: GVL.waterlevel
    Rectangle (416,432 100x20), "Soap level"
    Rectangle (516,432 45x20), "%d", text variable: GVL.soaplevel
    Rectangle (357,175 215x90)
    Lamp1 (402,177 20x20), variable: GVL.temp_error, style: Lamp-Lamp1-Red
    Rectangle (362,197 100x19), "Temperature error"
    Lamp1 (507,177 20x20), variable: GVL.bulls_eye_open, style: Lamp-Lamp1-Red
    Rectangle (467,197 100x19), "Door opened"
    Lamp1 (402,223 20x20), variable: GVL.prog_error, style: Lamp-Lamp1-Red
    Rectangle (362,243 100x19), "Program error"
    Lamp1 (507,223 20x20), variable: GVL.soap_alarm, style: Lamp-Lamp1-Red
    Rectangle (467,243 100x19), "Soap required"
    Rectangle (357,35 215x25), "FAULT PANEL"
    Rectangle (357,60 215x70)
    Rectangle (362,105 60x20), "Resistor"
    RockerSwitch (377,65 30x40), variable: GVL.heat_fail, behaviour: TOGGLE, style: Switch-RockerSwitch-Red
    RockerSwitch (449,65 30x40), variable: GVL.water_in_fail, behaviour: TOGGLE, style: Switch-RockerSwitch-Red
    Rectangle (434,105 60x20), "Intake"
    RockerSwitch (522,65 30x40), variable: GVL.water_out_fail, behaviour: TOGGLE, style: Switch-RockerSwitch-Red
    Rectangle (507,105 60x20), "Drain"
    Rectangle (357,271 215x25), "FAULT DETECTION"
    Rectangle (357,296 215x107)
    Lamp1 (367,299 30x30), variable: GVL.heat_alarm, style: Lamp-Lamp1-Red
    Rectangle (412,304 140x20), "Resistor fault detected"
    Lamp1 (367,370 30x30), variable: GVL.water_out_alarm, style: Lamp-Lamp1-Red
    Lamp1 (367,334 30x30), variable: GVL.water_in_alarm, style: Lamp-Lamp1-Red
    Rectangle (412,339 140x20), "Intake fault detected"
    Rectangle (412,375 140x20), "Drain fault detected"
    Rectangle (52,416 38x0)
        p2773130477: -GVL.soaplevel
    Rectangle (51,376 40x20), "SOAP"
    Polygon (65,280) (65,300) (52,300) (71,315) (90,300) (77,300) (77,280), colour toggle: GVL.fillsoap
        toggle GVL.fillsoap
    Rectangle (41,254 60x20), "PUT SOAP"
END_VISUALIZATION
